(* IEC 61131-3 sources: volt/packages/volt-lsp-iec/test-corpus/pro2193/Device/Plc Logic/Application/09 Misc/Library Manager/L_MC1P_MotionControlBasic (part 2) *)

(* ---- _AXIS_REF_ENC.pou ---- *)
FUNCTION_BLOCK _AXIS_REF_ENC EXTENDS _AXIS_REF_COM
VAR_INPUT
	DIENCODERPOSITION : DINT;
	XENCODERPOSVALID : BOOL := TRUE;
	POSSIGNALPROCESSING : L_MC1P_IPosSignalProcessing;
END_VAR
VAR
	WENCFILTERCYCLES : WORD := 1;
	WENCFILTERCYCLESPOS : WORD := 1;
	VELFILTER : L_MC1P_MeanValueFilter;
	ENCODERCONV : L_MC1P_EncoderConv;
	UDITOTALMEASURINGRANGE : UDINT := 4294967295;
	OPTPOSQUANT : L_MC1P_OptimizePosQuantisation;
	EXTRAPOLATION : L_MC1P_Extra_Interpolation;
	LRSETVALDELAYTIME : LREAL := 0;
	ECOMPENSATIONMODE : L_MC1P_CompensationMode := L_MC1P_CompensationMode.Off;
	XISABSOLUTEENCODER : BOOL := FALSE;
	XDRIVEENABLEDINTERN : BOOL;
	USIHOMEPOSPERMANTENTSETOLD : USINT;
	XHOMEPOSPERMANTENTSETFROMINTERN : BOOL;
	XENCODERPOSVALIDOLD : BOOL;
	XENCODERPOSVALIDINT : BOOL;
	XRESETENCODERPOSHANDLING : BOOL;
	WMICSECTICKSACT : WORD;
	WMICSECTICKSOLD : WORD;
	DIVELEXACT : DINT;
	XABSENCAVAILABLE : BOOL := FALSE;
	DWABSTIMERINFASTINPUTRESOLUTION : DWORD;
	XMANIPULATEABSCOUNTER : BOOL := FALSE;
	XCOUNTEROVERFLOW : BOOL;
	LRSCALEUNITTOPOSOLD : LREAL;
	XORIENTATIONINVACTOLD : BOOL;
	SCHOMEPARAMETER_LROFFSETPOSITIONOLD : LREAL;
	XMAXVELEXCEEDED : BOOL;
	XMAXVELEXCEEDEDOLD : BOOL;
	ITFENCODERPOSFILTER : L_MC1P_IEncoderPosFilter;
	ITFENCODERPOSFILTEROLD : L_MC1P_IEncoderPosFilter;
	ITFENCODERPOSFILTEREXTERNAL : L_MC1P_IEncoderPosFilter;
	FB_MEANPOSFILTER : L_MC1P_MeanEncoderPositionFilter;
	FB_BUTTERWORTHPOSFILTER : L_MC1P_ButterworthEncoderPosFilter;
	LRBTWFILTERTIME : LREAL;
	EENCINPUTFILTER : USINT;
	WENCFILTERCYCLESACTIVE : WORD;
	DIBTWFILTERTIME : DINT;
	EENCPOSFILTERSTATE : WORD;
	EENCVELFILTERSTATE : WORD;
	WENCODERPOSHANDLING : WORD;
	XTIMESTAMPFORPOSSUPPORTED : BOOL;
	_PTASKMAPLIST : POINTER TO IoStandard.IoConfigTaskMap;
	_NTASKMAPLISTCOUNT : DINT;
	_WMODULETYPE : UINT;
	_DWINSTANCE : UDINT;
	_CONNECTOR : POINTER TO IoConfigConnector;
	EENCODERTYPE : L_Mc1P_EncoderType;
	DIINPUTPOSOLD : DINT;
	DIACTPOSUNFILTERED : DINT;
	LRRESIDUALPOSUNFILTERED : LREAL;
	XCONFIGCHANGED : BOOL;
	DWPOSTIMESTAMP : DWORD;
	POSSIGNALPROCESSINGINT : L_MC1P_PosSignalProcessing;
	XSSIENCODER : BOOL := FALSE;
	DWENCODERUPDATETIME : DWORD;
	DIACTPOS1616 : DINT;
	XACTVELFROMPOS : BOOL;
	PDWABSOLUTECOUNTERINT : POINTER TO DWORD;
	DIACTPOSRAWOLD : DINT;
	XVELEXACTSUPPORTED : BOOL;
	CMPID_CMP_LSMCFREEENCODER : DWORD := 16#1028200D;
	ENCHOMEPOSPERMANTENTSETACTIVE : BOOL;
	GETTIMEREFVALUE : DWORD;
	HOMEPOSPERMANTENTSETACTIVE : BOOL;
	WAITFORAXISDETECTION : BOOL;
END_VAR
END_FUNCTION_BLOCK

METHOD CALCACTPOSFROMHWCOUNTER : LREAL
END_METHOD

METHOD CALCACTPOSUNFILTERED : LREAL
END_METHOD

METHOD CALCACTVALUES
END_METHOD

METHOD CALCEXTRAPOLATIONVALUES
VAR_INPUT
	LRACTPOSIN : LREAL;
	LRACTVELIN : LREAL;
	LRACTACCIN : LREAL;
	LRACTTORQUEIN : LREAL;
END_VAR
VAR_OUTPUT
	LRACTPOSOUT : LREAL;
	LRACTVELOUT : LREAL;
	LRACTACCOUT : LREAL;
	LRACTTORQUEOUT : LREAL;
END_VAR
END_METHOD

METHOD CALLRECIEVEPARAMETER
END_METHOD

METHOD CHECKPLAUSIBILITYOFACTVALUES
END_METHOD

METHOD ENCODERSIGNALHANDLING : BOOL
END_METHOD

METHOD GETACTVELOCITYEXACT : LREAL
END_METHOD

METHOD PREPAREINPUTDATA : BOOL
END_METHOD

METHOD READENCODERINPUT : BOOL
VAR_INPUT
	DINEWENCPOS : DINT;
END_VAR
END_METHOD

METHOD RESETACTPOS
END_METHOD

METHOD RESETAXISCONNECTOR
END_METHOD

METHOD RESETENCODERVALUES
END_METHOD

METHOD SETENCODERFILTERINTERFACE
VAR_INPUT
	IENCODERFILTERITF : L_MC1P_IEncoderPosFilter;
END_VAR
END_METHOD

METHOD SETHOMEPOSITION2
VAR_INPUT
	POSITION : LREAL;
	RELATIVE : BOOL;
	XRESTARTPOSITIONING : BOOL := FALSE;
	EHOMEPOSINFO : L_IE1P_Error;
END_VAR
END_METHOD

METHOD ENCNEWHOMEPOSLOADED : BOOL
VAR_INPUT
	DWCALLYCLE : DWORD;
	DWDELAY : DWORD;
END_VAR
END_METHOD

METHOD ENCRESETACTPOS
END_METHOD

METHOD ENCRESETHOMEPOS
VAR_INPUT
	ERESETINFO : L_IE1P_Error;
END_VAR
END_METHOD

METHOD ENCSETHOMEPOSITION
VAR_INPUT
	POSITION : LREAL;
	RELATIVE : BOOL;
	POSDIFF : LREAL;
	EHOMEPOSINFO : L_IE1P_Error;
END_VAR
END_METHOD

METHOD ENCSIGNALVALID : BOOL
VAR_OUTPUT
	XSIGNALVALIDOLD : BOOL;
	EENCERRORID : L_IE1P_Error;
END_VAR
END_METHOD

METHOD GETACTPOSINCR : DINT
END_METHOD

METHOD GETACTPOSINCR1616 : DINT
END_METHOD

METHOD GETACTVALUES
VAR_OUTPUT
	LRACTPOS : LREAL;
	LRACTVEL : LREAL;
	LRACTACC : LREAL;
	LRACTPOSUNFILTERED : LREAL;
	LRACTPOSROUNDS : LREAL;
END_VAR
END_METHOD

METHOD GETAXISINSTANCE : POINTER TO _AXIS_REF_REAL
END_METHOD

METHOD GETCONFIGCHANGED : BOOL
END_METHOD

METHOD GETENCODERINTERFACE : L_MC1P_IEncoderInterface
END_METHOD

METHOD GETHOMEPOSAVAILABLE : BOOL
END_METHOD

METHOD SETHOMEPOSAVAILABLE
VAR_INPUT
	XHOMEPOSAVAILABLE : BOOL;
END_VAR
END_METHOD

METHOD GETVIRTUAL : BOOL
END_METHOD

METHOD CALCSCALEFUNCTIONS
VAR_INPUT
	OFFSET : DWORD;
	INDEX : WORD;
END_VAR
END_METHOD

METHOD CALLTRANSMITPARAMETER
END_METHOD

METHOD PDCONVACTPOS : DINT
VAR_INPUT
	DIINPUT : DINT;
END_VAR
END_METHOD

METHOD PDCONVACTPOSENCCONV : DINT
VAR_INPUT
	DIINPUT : DINT;
END_VAR
END_METHOD

METHOD PDCONVACTVEL : DINT
VAR_INPUT
	DIINPUT : DINT;
END_VAR
END_METHOD

METHOD PDHANDLETIMESTAMPS : DINT
VAR_INPUT
	WMICSECTICK : WORD;
END_VAR
END_METHOD

METHOD CONFIGUREAXIS
END_METHOD

METHOD CONNECTMOTIONUTILS
VAR_INPUT
	DRIVEUTILS : L_MC1P_IDriveUtils;
	AXISEXTENSION : L_MC1P_IAxisExtension;
END_VAR
END_METHOD

METHOD CALCAFTERREADINPUTS : INT
END_METHOD

METHOD CALCBEFOREREADINPUTS : INT
END_METHOD

METHOD CALCBEFOREWRITEOUTPUTS : INT
END_METHOD

METHOD FB_INIT : BOOL
VAR_INPUT
	BINITRETAINS : BOOL;
	BINCOPYCODE : BOOL;
END_VAR
END_METHOD

METHOD IODRVUPDATEMAPPING : UDINT
VAR_INPUT
	PTASKMAPLIST : POINTER TO IoConfigTaskMap;
	NCOUNT : DINT;
END_VAR
END_METHOD

METHOD INITIALIZE : UDINT
VAR_INPUT
	WMODULETYPE : UINT;
	DWINSTANCE : UDINT;
	PCONNECTOR : POINTER TO IoConfigConnector;
END_VAR
END_METHOD

(* ---- _AXIS_REF_ENC_BPB.pou ---- *)
FUNCTION_BLOCK _AXIS_REF_ENC_BPB EXTENDS _AXIS_REF_ENC
VAR
	AXISEXTENSION : L_MC1P_AxisExtension_EncBPB;
	MOTIONUTILS : L_MC1P_MotionUtils_EncBPB;
END_VAR
END_FUNCTION_BLOCK

METHOD FB_INIT : BOOL
VAR_INPUT
	BINITRETAINS : BOOL;
	BINCOPYCODE : BOOL;
END_VAR
END_METHOD

(* ---- _AXIS_REF_ENC_FREE.pou ---- *)
FUNCTION_BLOCK _AXIS_REF_ENC_FREE EXTENDS _AXIS_REF_ENC
VAR
	AXISEXTENSION : L_MC1P_AxisExtension_EncFree;
	MOTIONUTILS : L_MC1P_MotionUtils_EncFree;
END_VAR
END_FUNCTION_BLOCK

METHOD FB_INIT : BOOL
VAR_INPUT
	BINITRETAINS : BOOL;
	BINCOPYCODE : BOOL;
END_VAR
END_METHOD

(* ---- _AXIS_REF_ENC_I500_ECAT.pou ---- *)
FUNCTION_BLOCK _AXIS_REF_ENC_I500_ECAT EXTENDS _AXIS_REF_ENC
VAR
	AXISEXTENSION : L_MC1P_AxisExtension_Enci500;
	MOTIONUTILS : L_MC1P_MotionUtils_Enci500;
END_VAR
END_FUNCTION_BLOCK

METHOD FB_INIT : BOOL
VAR_INPUT
	BINITRETAINS : BOOL;
	BINCOPYCODE : BOOL;
END_VAR
END_METHOD

(* ---- _AXIS_REF_ENC_I900.pou ---- *)
FUNCTION_BLOCK _AXIS_REF_ENC_I900 EXTENDS _AXIS_REF_ENC
END_FUNCTION_BLOCK

METHOD HLP_INITPARREF
END_METHOD

METHOD HLP_READPARAMETER : BOOL
VAR_INPUT
	PARAMETER : DINT;
	PLRVALUE : POINTER TO LREAL;
END_VAR
END_METHOD

(* ---- _AXIS_REF_ENC_I900_CIA.pou ---- *)
FUNCTION_BLOCK _AXIS_REF_ENC_I900_CIA EXTENDS _AXIS_REF_ENC_i900_Target
END_FUNCTION_BLOCK

METHOD SETDRIVECONFIG
VAR_OUTPUT
	XDONE : BOOL;
	XERROR : BOOL;
	WERRORID : WORD;
END_VAR
END_METHOD

METHOD CALCULATESCALING : BOOL
END_METHOD

METHOD FB_INIT : BOOL
VAR_INPUT
	BINITRETAINS : BOOL;
	BINCOPYCODE : BOOL;
END_VAR
END_METHOD

(* ---- _AXIS_REF_ENC_I900_ECAT.pou ---- *)
FUNCTION_BLOCK _AXIS_REF_ENC_I900_ECAT EXTENDS _AXIS_REF_ENC
VAR
	AXISEXTENSION : L_MC1P_AxisExtension_Enci900_ECAT;
	MOTIONUTILS : L_Mc1P_MotionUtils_Enci900_ECAT;
	RETAINMANAGEMENT : L_MC1P_MotionUtilsRetainHandling;
END_VAR
END_FUNCTION_BLOCK

METHOD FB_INIT : BOOL
VAR_INPUT
	BINITRETAINS : BOOL;
	BINCOPYCODE : BOOL;
END_VAR
END_METHOD

(* ---- _AXIS_REF_ENC_I900_TARGET.pou ---- *)
FUNCTION_BLOCK _AXIS_REF_ENC_I900_TARGET EXTENDS _AXIS_REF_ENC_i900
VAR
	AXISEXTENSION : L_MC1P_AxisExtension_Enci900_Target;
	MOTIONUTILS : L_MC1P_MotionUtils_Enci900_Target;
	RETAINMANAGEMENT : L_MC1P_MotionUtilsRetainHandling;
END_VAR
END_FUNCTION_BLOCK

METHOD CALLRECIEVEPARAMETER
END_METHOD

METHOD CONFIGUREAXISCONNECTOR
END_METHOD

METHOD GETIECADRESS
END_METHOD

METHOD FB_INIT : BOOL
VAR_INPUT
	BINITRETAINS : BOOL;
	BINCOPYCODE : BOOL;
END_VAR
END_METHOD

(* ---- _AXIS_REF_ENC_IO_ETC.pou ---- *)
FUNCTION_BLOCK _AXIS_REF_ENC_IO_ETC EXTENDS _AXIS_REF_ENC
VAR
	AXISEXTENSION : L_MC1P_AxisExtension_EncIOEtc;
	MOTIONUTILS : L_MC1P_MotionUtils_EncIOEtc;
END_VAR
END_FUNCTION_BLOCK

METHOD INITIALIZE : UDINT
VAR_INPUT
	WMODULETYPE : UINT;
	DWINSTANCE : UDINT;
	PCONNECTOR : POINTER TO IoConfigConnector;
END_VAR
END_METHOD

METHOD FB_INIT : BOOL
VAR_INPUT
	BINITRETAINS : BOOL;
	BINCOPYCODE : BOOL;
END_VAR
END_METHOD

(* ---- _AXIS_REF_ENC_UNIVERSAL.pou ---- *)
FUNCTION_BLOCK _AXIS_REF_ENC_UNIVERSAL EXTENDS _AXIS_REF_ENC
VAR
	FBDRIVESPECIFIC : L_MC1P_DriveSpecific_Enc_Free;
	AXISEXTENSIONFACTORY : L_MC1P_UniversalEncoderFactory;
	ITFDRIVEUTILSTOCONNECT : POINTER TO L_MC1P_IDriveUtils;
	ITFAXISEXTENSION : L_MC1P_IAxisExtension;
	UITYPE : UINT := 2;
	DRIVESPECIFICBASIC : L_MC1P_IDriveSpecificImplBase;
	WAITFORAXISDETECTION : BOOL;
END_VAR
END_FUNCTION_BLOCK

METHOD CALCAFTERREADINPUTS : INT
END_METHOD

METHOD CONNECTASYNC : BOOL
END_METHOD

METHOD CREATEAXISEXTENSION : L_MC1P_IAxisExtension
VAR_INPUT
	EAXISEXTENSIONTYPE : L_MC1P_AxisExtensionTypes;
END_VAR
END_METHOD

METHOD DISCONNECTMOTIONUTILS : BOOL
VAR_INPUT
	EDISCONNECTMODE : L_IF1P_DisconnectMode;
END_VAR
END_METHOD

METHOD FINDANDCONNECTMOTIONUTILS
END_METHOD

METHOD FINDDRIVEUTILSINMOTIONCONNECTOR : BOOL
VAR_INPUT
	PECATSLAVECONNECTOR : POINTER TO IoConfigConnector;
	SUBDEVICE : UINT;
END_VAR
END_METHOD

METHOD INITIALIZE : UDINT
VAR_INPUT
	WMODULETYPE : UINT;
	DWINSTANCE : UDINT;
	PCONNECTOR : POINTER TO IoConfigConnector;
END_VAR
END_METHOD

METHOD FB_INIT : BOOL
VAR_INPUT
	BINITRETAINS : BOOL;
	BINCOPYCODE : BOOL;
END_VAR
END_METHOD

METHOD CONNECTDEVICE : UINT
VAR_INPUT
	DEVICEMODULEHANDLER : L_IMHP_IModuleHandler;
	UISUBDEVICE : UINT := 0;
	EDISCONNECTMODE : L_IF1P_DisconnectMode;
	XDISCONNECTEXISTINGCONNECTION : BOOL;
END_VAR
VAR_OUTPUT
	ITFCONNECTIONFBSTATUS : L_IF1P_IStatus;
END_VAR
END_METHOD

METHOD DISCONNECTDEVICE : UINT
VAR_INPUT
	EDISCONNECTMODE : L_IF1P_DisconnectMode;
	XBUSYBEFORE : BOOL;
END_VAR
VAR_OUTPUT
	ITFCONNECTIONFBSTATUS : L_IF1P_IStatus;
END_VAR
END_METHOD

METHOD GEFUNCTIONTINSTANCEPOINTER : POINTER TO BYTE
END_METHOD

METHOD GETCONNECTEDDEVICE : L_IMHP_IModuleHandler
VAR_OUTPUT
	UISUBDEVICE : UINT := 0;
	XVALID : BOOL;
	ITFCONNECTIONFBSTATUS : L_IF1P_IStatus;
END_VAR
END_METHOD

METHOD GETCONNECTIONDIAGNOSTIC
VAR_OUTPUT
	WUSEDBY_COMP : WORD;
	WUSEDBY_SUBCOMP : WORD;
	WACTIVEMODE : WORD;
	WSUBDEVICE : WORD;
	SCONNECTIONSOURE : STRING;
END_VAR
END_METHOD

METHOD GETITFCONNECTSTATUS
VAR_OUTPUT
	ITFCONNECTIONFBSTATUS : L_IF1P_IStatus;
END_VAR
END_METHOD

(* ---- _AXIS_REF_GENERIC.pou ---- *)
FUNCTION_BLOCK _AXIS_REF_GENERIC EXTENDS _AXIS_REF_COM
VAR
	AXISEXTENSION : L_MC1P_AxisExtension_GenericDrive;
	MOTIONUTILS : L_MC1P_MotionUtils_GenericDrive;
	RETAINMANAGEMENT : L_MC1P_MotionUtilsRetainHandling;
END_VAR
END_FUNCTION_BLOCK

METHOD SETGENERICCONFIGURATION
VAR_INPUT
	ITFGENERICCONFIG : L_MC1P_IGenericAxisConfiguration;
END_VAR
END_METHOD

METHOD FB_INIT : BOOL
VAR_INPUT
	BINITRETAINS : BOOL;
	BINCOPYCODE : BOOL;
END_VAR
END_METHOD

(* ---- _AXIS_REF_I500.pou ---- *)
FUNCTION_BLOCK _AXIS_REF_I500 EXTENDS _AXIS_REF_COM
VAR
	CONFIGAXIS : L_MC1P_Config_i500;
	FBEXTENDEDMAPPINGACCESS : L_MC1P_ExtendedMappingAccess;
	BRAKE : L_MC1P_BrakeControl;
	WNETWORDIN1 : REFERENCE TO WORD;
	WNETWORDIN2 : REFERENCE TO WORD;
	WNETWORDIN3 : REFERENCE TO WORD;
	WNETWORDIN4 : REFERENCE TO WORD;
	WNETWORDOUT1 : REFERENCE TO WORD;
	WNETWORDOUT2 : REFERENCE TO WORD;
	PXDUMMY : POINTER TO BOOL;
	XENABLEDRIVEOLD : BOOL;
	XDEACTIVATEPOSCTRLEXTENCERROR : BOOL;
	NETWORDIN1 : WORD;
	NETWORDIN2 : WORD;
	NETWORDIN3 : WORD;
	NETWORDIN4 : WORD;
	NETWORDOUT1 : WORD;
	NETWORDOUT2 : WORD;
END_VAR
END_FUNCTION_BLOCK

(* ---- _AXIS_REF_I500_CAN.pou ---- *)
FUNCTION_BLOCK _AXIS_REF_I500_CAN EXTENDS _AXIS_REF_i500
VAR
	AXISEXTENSION : L_MC1P_AxisExtension_i500_CAN;
	MOTIONUTILS : L_MC1P_MotionUtils_i500_CAN;
END_VAR
END_FUNCTION_BLOCK

METHOD FB_INIT : BOOL
VAR_INPUT
	BINITRETAINS : BOOL;
	BINCOPYCODE : BOOL;
END_VAR
END_METHOD

(* ---- _AXIS_REF_I500_ETC.pou ---- *)
FUNCTION_BLOCK _AXIS_REF_I500_ETC EXTENDS _AXIS_REF_i500
VAR
	AXISEXTENSION : L_MC1P_AxisExtension_i500_ECAT;
	MOTIONUTILS : L_MC1P_MotionUtils_i500_ECAT;
END_VAR
END_FUNCTION_BLOCK

METHOD FB_INIT : BOOL
VAR_INPUT
	BINITRETAINS : BOOL;
	BINCOPYCODE : BOOL;
END_VAR
END_METHOD

(* ---- _AXIS_REF_I700.pou ---- *)
FUNCTION_BLOCK _AXIS_REF_I700 EXTENDS _AXIS_REF_COM
VAR
	XSLOT2 : BOOL;
	AXISEXTENSION : L_MC1P_AxisExtension_i700;
	MOTIONUTILS : L_MC1P_MotionUtils_i700;
	RETAINMANAGEMENT : L_MC1P_MotionUtilsRetainHandling;
END_VAR
END_FUNCTION_BLOCK

METHOD INITIALIZE : UDINT
VAR_INPUT
	WMODULETYPE : UINT;
	DWINSTANCE : UDINT;
	PCONNECTOR : POINTER TO IoConfigConnector;
END_VAR
END_METHOD

METHOD FB_INIT : BOOL
VAR_INPUT
	BINITRETAINS : BOOL;
	BINCOPYCODE : BOOL;
END_VAR
END_METHOD

(* ---- _AXIS_REF_I700_SLOT1.pou ---- *)
FUNCTION_BLOCK _AXIS_REF_I700_SLOT1 EXTENDS _AXIS_REF_i700
END_FUNCTION_BLOCK

METHOD FB_INIT : BOOL
VAR_INPUT
	BINITRETAINS : BOOL;
	BINCOPYCODE : BOOL;
END_VAR
END_METHOD

(* ---- _AXIS_REF_I750.pou ---- *)
FUNCTION_BLOCK _AXIS_REF_I750 EXTENDS _AXIS_REF_COM
VAR
	XSLOT2 : BOOL;
	AXISEXTENSION : L_MC1P_AxisExtension_i750;
	MOTIONUTILS : L_MC1P_MotionUtils_i750;
	RETAINMANAGEMENT : L_MC1P_MotionUtilsRetainHandling;
END_VAR
END_FUNCTION_BLOCK

METHOD FB_INIT : BOOL
VAR_INPUT
	BINITRETAINS : BOOL;
	BINCOPYCODE : BOOL;
END_VAR
END_METHOD

(* ---- _AXIS_REF_I900.pou ---- *)
FUNCTION_BLOCK _AXIS_REF_I900 EXTENDS _AXIS_REF_COM
VAR
	XSLOT2 : BOOL;
	AXISEXTENSION : L_MC1P_AxisExtension_i950;
	MOTIONUTILS : L_MC1P_MotionUtils_i950;
	RETAINMANAGEMENT : L_MC1P_MotionUtilsRetainHandling;
END_VAR
END_FUNCTION_BLOCK

METHOD FB_INIT : BOOL
VAR_INPUT
	BINITRETAINS : BOOL;
	BINCOPYCODE : BOOL;
END_VAR
END_METHOD

(* ---- _AXIS_REF_I900_CIAADV.pou ---- *)
FUNCTION_BLOCK _AXIS_REF_I900_CIAADV EXTENDS _AXIS_REF_COM
VAR
	XSLOT2 : BOOL;
	AXISEXTENSION : L_MC1P_AxisExtension_i950_CiaAdv;
	MOTIONUTILS : L_MC1P_MotionUtils_i950_CiaAdv;
	RETAINMANAGEMENT : L_MC1P_MotionUtilsRetainHandling;
END_VAR
END_FUNCTION_BLOCK

METHOD FB_INIT : BOOL
VAR_INPUT
	BINITRETAINS : BOOL;
	BINCOPYCODE : BOOL;
END_VAR
END_METHOD

(* ---- _AXIS_REF_I900_DRIVE.pou ---- *)
FUNCTION_BLOCK _AXIS_REF_I900_DRIVE EXTENDS _AXIS_REF_COM
VAR
	LRHOMETORQUELIMIT : LREAL;
	LRHOMETORQUELIMITTIME : LREAL;
	EFOLLOWINGERRORREACTIONI900 : USINT;
	XIGNOREPDOINTERFACEDISABLED : BOOL := FALSE;
	INTERPOLATION : L_MC1P_DelaySetValues2;
	LRSETVALDELAYTIME : LREAL := 0;
	ECOMPENSATIONMODE : L_MC1P_CompensationMode := L_MC1P_CompensationMode.Off;
	UIPOSCTRLADAPTACTIVEVALUE : UINT;
	USIPOSCTRLADAPTIONFROM0X2985 : USINT := 0;
	POSCTRLADAPTIONCURVE : L_MC1P_PosCtrlAdaptionCurve;
	DWCOMPATIBILITYFLAGS_0X2DE0_28 : DWORD;
	WAITFORAXISDETECTION : BOOL;
END_VAR
END_FUNCTION_BLOCK

METHOD GETACTIVEPOSCTRLADAPTVALUE : LREAL
END_METHOD

METHOD CONFIGUREAXISCONNECTOR
END_METHOD

METHOD CALCSCALEFUNCTIONS
VAR_INPUT
	OFFSET : DWORD;
	INDEX : WORD;
END_VAR
END_METHOD

METHOD UPDATEDRIVEOFFSETHANDLING
VAR_INPUT
	DWACTCYCLECOUNTERVALUE : DWORD;
	XRESET : BOOL;
END_VAR
END_METHOD

METHOD HLP_INITPARREF
END_METHOD

METHOD HLP_READBOOLPARAMETER : BOOL
VAR_INPUT
	PARAMETER : DINT;
	PXVALUE : POINTER TO BOOL;
END_VAR
END_METHOD

METHOD HLP_READPARAMETER : BOOL
VAR_INPUT
	PARAMETER : DINT;
	PLRVALUE : POINTER TO LREAL;
END_VAR
END_METHOD

METHOD HLP_WRITEBOOLPARAMETER : BOOL
VAR_INPUT
	PARAMETER : DINT;
	PXVALUE : POINTER TO BOOL;
END_VAR
VAR_OUTPUT
	WERRORID : WORD;
END_VAR
END_METHOD

METHOD CALCBEFOREREADINPUTS : INT
END_METHOD

METHOD CALCBEFOREWRITEOUTPUTS : INT
END_METHOD

METHOD FB_INIT : BOOL
VAR_INPUT
	BINITRETAINS : BOOL;
	BINCOPYCODE : BOOL;
END_VAR
END_METHOD

(* ---- _AXIS_REF_I900_DRIVE_CIA.pou ---- *)
FUNCTION_BLOCK _AXIS_REF_I900_DRIVE_CIA EXTENDS _AXIS_REF_i900_Drive_Target
VAR_INPUT
	XOPMODEVIACIA402INTERFACE : BOOL;
	XCONTROLVIACIAINTERFACE : BOOL;
	XSETVALUESVIAAPPLICATION : BOOL;
	CIA_CTRL_EXT : WORD;
	CIA_OPMOD_EXT : SINT;
	WLENZECTRL_EXT : WORD;
	WTPCONTROL12 : WORD;
	WTPCONTROL34 : WORD;
	XCONTROLVIACIAINTERFACEOLD : BOOL;
	XEXTSETVALUESVALID : BOOL;
	LRSETPOSITION_EXT : LREAL;
	LRSETVELOCITY_EXT : LREAL;
	LRSETTORQUE_EXT : LREAL;
	LRSETVELOCITYLIMITHIGH_EXT : LREAL;
	LRSETVELOCITYLIMITLOW_EXT : LREAL;
	LRSETVLVELOCITY_EXT : LREAL;
END_VAR
VAR_OUTPUT
	WTPSTATUS12 : WORD;
	WTPSTATUS34 : WORD;
	LRTP1_POSEDGE : LREAL;
	LRTP1_NEGEDGE : LREAL;
	DWTP1_TIMENEGEDGE : DWORD;
	DWTP1_TIMEPOSEDGE : DWORD;
	LRTP2_POSEDGE : LREAL;
	LRTP2_NEGEDGE : LREAL;
	DWTP2_TIMENEGEDGE : DWORD;
	DWTP2_TIMEPOSEDGE : DWORD;
	LRTP3_POSEDGE : LREAL;
	LRTP3_NEGEDGE : LREAL;
	DWTP3_TIMENEGEDGE : DWORD;
	DWTP3_TIMEPOSEDGE : DWORD;
	LRTP4_POSEDGE : LREAL;
	LRTP4_NEGEDGE : LREAL;
	DWTP4_TIMENEGEDGE : DWORD;
	DWTP4_TIMEPOSEDGE : DWORD;
	LRACTCONTROLEFFORT : LREAL;
END_VAR
VAR
	WPOWID : WORD;
	CIA_CTRLOLD_EXT : WORD;
	XSETVALUESVIAAPPLICATION_INT : BOOL;
	XINTTP1ACTIVE : BOOL;
	XINTTP2ACTIVE : BOOL;
	XINTTP3ACTIVE : BOOL;
	XINTTP4ACTIVE : BOOL;
	DIDRIVEREFOFFSET : DINT;
	DIDRIVEREFOFFSETABS : DINT;
	DIDRIVEREFOFFSETABSOLD : DINT;
	XDRIVELOADPOS : BOOL;
	XIGNOREDRIVEOFFSET : BOOL;
	DIDEBUGPOS : DINT;
	REFOFFSETHANDLING : L_MC1P_i900RefOffsetHandling;
	XREFOFFSETHANDLINGCALCULATED : BOOL;
	XCONFIGCHANGED : BOOL;
	XCONFIGCHANGEDENCODER : BOOL;
	X2NDFDBACTIVE : BOOL;
	X2NDFDBOBSERVATIONACTIVE : BOOL;
	LRDIRECTIONHYSTERESISDIFFOLD : LREAL;
	LRACTCONTROLEFFORTDRIVE : LREAL;
	WLENZECTRL : REFERENCE TO WORD;
	LRSPEEDCTRLINT : REFERENCE TO LREAL;
	XNEWHOMEPOSHANDLINGCIA402ADV : BOOL;
	CIA402ADVANCEDAXIS : BOOL;
	STARTPOSFORINTERNALSTOP : LREAL;
END_VAR
END_FUNCTION_BLOCK

METHOD CALCACTVALUES
END_METHOD

METHOD CALCCONTOLLER
END_METHOD

METHOD CALCDRIVEHOMEOFFSET : DINT
VAR_INPUT
	LROLDPOS : LREAL;
	LRNEWPOSPOS : LREAL;
END_VAR
END_METHOD

METHOD CHECKFOLLOWINGERROR : BOOL
END_METHOD

METHOD CHECKPLNOTVALID : BOOL
END_METHOD

METHOD CONVERTTPPOSAPP : LREAL
VAR_INPUT
	DIPOS : DINT;
END_VAR
END_METHOD

METHOD ENABLEDRIVE : BOOL
VAR_INPUT
	XENABLE : BOOL;
END_VAR
END_METHOD

METHOD GETACTDIRECTION : MC_DIRECTION
VAR_INPUT
	XCALCULATE : BOOL;
END_VAR
END_METHOD

METHOD GETDRIVESTATE : BOOL
END_METHOD

METHOD HANDLETPCONTROL
VAR_INPUT
	WTPCONTROL : WORD;
	PWCONTROL : POINTER TO WORD;
END_VAR
VAR_IN_OUT
	XTP1ACTIVE : BOOL;
	XTP2ACTIVE : BOOL;
END_VAR
END_METHOD

METHOD RESETACTPOS
END_METHOD

METHOD RESETCONFIGCHANGED
END_METHOD

METHOD SETHOMEPOSITION2
VAR_INPUT
	POSITION : LREAL;
	RELATIVE : BOOL;
	XRESTARTPOSITIONING : BOOL := FALSE;
	EHOMEPOSINFO : L_IE1P_Error;
END_VAR
END_METHOD

METHOD PDCONVACTPOS : DINT
VAR_INPUT
	DIINPUT : DINT;
END_VAR
END_METHOD

METHOD PDCONVSETPOS : DINT
VAR_INPUT
	XSETEQACTONDISABLED : BOOL;
END_VAR
END_METHOD

METHOD PDCONVTPPOS : DINT
VAR_INPUT
	DIPOS : DINT;
END_VAR
END_METHOD

METHOD SETDRIVECONFIG
VAR_OUTPUT
	XDONE : BOOL;
	XERROR : BOOL;
	WERRORID : WORD;
END_VAR
END_METHOD

METHOD CALCPOSTOUNIT : LREAL
VAR_INPUT
	DIPOSITION : DINT;
END_VAR
END_METHOD

METHOD CALCRPMTOUNIT : LREAL
VAR_INPUT
	ISPEED : INT;
END_VAR
END_METHOD

METHOD CALCSPEEDTOUNIT : LREAL
VAR_INPUT
	DISPEED : DINT;
END_VAR
END_METHOD

METHOD CALCTORQUETOUNIT : LREAL
VAR_INPUT
	ITORQUE : INT;
END_VAR
END_METHOD

METHOD CALCUNITTOPOS : DINT
VAR_INPUT
	LRPOSITION : LREAL;
END_VAR
END_METHOD

METHOD CALCUNITTORPM : INT
VAR_INPUT
	LRVELOCITY : LREAL;
END_VAR
END_METHOD

METHOD CALCUNITTOSPEED : DINT
VAR_INPUT
	LRVELOCITY : LREAL;
END_VAR
END_METHOD

METHOD CALCUNITTOTORQUE : INT
VAR_INPUT
	LRTORQUE : LREAL;
END_VAR
END_METHOD

METHOD CALCULATESCALING : BOOL
END_METHOD

METHOD RESTOREACTPOS
VAR_INPUT
	PPOSDATA : POINTER TO L_MC1P_uRetainData;
END_VAR
END_METHOD

METHOD RETAINHANDLING : BOOL
END_METHOD

METHOD STOREACTPOS
VAR_INPUT
	PPOSDATA : POINTER TO L_MC1P_uRetainData;
END_VAR
END_METHOD

METHOD STOREADDITIONALRETAINDATA
VAR_INPUT
	PDATA : POINTER TO L_MC1P_uRetainData;
END_VAR
END_METHOD

METHOD CALCBEFOREREADINPUTS : INT
END_METHOD

METHOD GETIECADRESS
END_METHOD

METHOD RECEIVEPARAMETER2
VAR_INPUT
	WPARAMETER : WORD;
	PADRESS : POINTER TO BYTE;
	WSIZE : WORD;
	PADDDATA : POINTER TO L_SI9P_IODrvMappingData;
END_VAR
END_METHOD

METHOD RECEIVEPARAMETERCALC2
VAR_IN_OUT
	DATA : ARRAY [1..L_MC1P_Constants.gc_Rec_MaxDataIndex] OF POINTER TO L_MC1P_MappedElement;
END_VAR
END_METHOD

METHOD TRANSMITPARAMETER
VAR_INPUT
	WPARAMETER : WORD;
	PADRESS : POINTER TO BYTE;
	WSIZE : WORD;
END_VAR
END_METHOD

METHOD TRANSMITPARAMETER2
VAR_INPUT
	WPARAMETER : WORD;
	PADRESS : POINTER TO BYTE;
	WSIZE : WORD;
	PADDDATA : POINTER TO L_SI9P_IODrvMappingData;
END_VAR
END_METHOD

METHOD TRANSMITPARAMETERCALC2
VAR_IN_OUT
	DATA : ARRAY [1..L_MC1P_Constants.gc_Trans_MaxDataIndex] OF POINTER TO L_MC1P_MappedElement;
END_VAR
END_METHOD

METHOD FB_INIT : BOOL
VAR_INPUT
	BINITRETAINS : BOOL;
	BINCOPYCODE : BOOL;
END_VAR
END_METHOD

(* ---- _AXIS_REF_I900_DRIVE_TARGET.pou ---- *)
FUNCTION_BLOCK _AXIS_REF_I900_DRIVE_TARGET EXTENDS _AXIS_REF_i900_Drive
VAR
	AXISEXTENSION : L_MC1P_AxisExtension_i950_Drive;
	MOTIONUTILS : L_MC1P_MotionUtils_i950_Drive;
	RETAINMANAGEMENT : L_MC1P_MotionUtilsRetainHandling;
	ADWINTERNALMAPPEDWRITEOBJECTS : ARRAY [1..c_wMaxTransElem] OF DWORD;
	HEVENTSETERRORREACTION : SysTypes.RTS_IEC_HANDLE := SysTypes.RTS_INVALID_HANDLE;
	HINTERFACESETERRORREACTION : SysTypes.RTS_IEC_HANDLE := SysTypes.RTS_INVALID_HANDLE;
	HEVENTUPDATEACTIVEERROR : SysTypes.RTS_IEC_HANDLE := SysTypes.RTS_INVALID_HANDLE;
	HINTERFACEUPDATEACTIVEERROR : SysTypes.RTS_IEC_HANDLE := SysTypes.RTS_INVALID_HANDLE;
	XINITIALREADERRORSTATUS : BOOL := FALSE;
	USIACTIVEERRORINFO : USINT := 0;
	DWLEMERRORCODE : ARRAY [0..2] OF DWORD;
	USILEMSEVERITY : ARRAY [0..2] OF USINT;
	DWPARMONITID : DWORD;
	PIPARQSPOPTION : POINTER TO INT;
	PWPARQSPOPTIONVALID : POINTER TO WORD;
	IPARQSPOPTIONOLD : INT;
	PWPARMOTORRATEDSPEED : POINTER TO WORD;
	PWPARMOTORRATEDSPEEDVALID : POINTER TO WORD;
	WPARMOTORRATEDSPEEDOLD : WORD;
	PDWPARREFTORQUE : POINTER TO DWORD;
	PWPARREFTORQUEVALID : POINTER TO WORD;
	DWPARREFTORQUEOLD : DWORD;
	PDWPARINERTIAMOTOR : POINTER TO DWORD;
	PWPARINERTIAMOTORVALID : POINTER TO WORD;
	DWPARINERTIAMOTOROLD : DWORD;
	PUSIPARMCTRLMODE : POINTER TO USINT;
	PWPARMCTRLMODEVALID : POINTER TO WORD;
	USIPARMCTRLMODEOLD : USINT;
	PDWPARMOTORRATEDCURRENT : POINTER TO DWORD;
	PWPARMOTORRATEDCURRENTVALID : POINTER TO WORD;
	DWPARMOTORRATEDCURRENTOLD : DWORD;
	PDWPARCOMPATIBILITYMODE : POINTER TO DWORD;
	PWPARCOMPATIBILITYMODEVALID : POINTER TO WORD;
	DWPARCOMPATIBILITYMODEOLD : DWORD;
	APWPARGAINADAPTSPEED : ARRAY [1..5] OF POINTER TO WORD;
	APWPARGAINADAPTSPEEDVALID : ARRAY [1..5] OF POINTER TO WORD;
	APWPARGAINADAPTOUT : ARRAY [1..5] OF POINTER TO WORD;
	APWPARGAINADAPTOUTVALID : ARRAY [1..5] OF POINTER TO WORD;
	EQUICKSTOPOPTIONACTIVE : L_MC1P_QuickStopOption := L_MC1P_QuickStopOption.StayInQSP;
END_VAR
END_FUNCTION_BLOCK

METHOD CALCDEPENDENTTORQUEVALUES
VAR_INPUT
	DWDATA : DWORD;
END_VAR
END_METHOD

METHOD GETACTIVEQUICKSTOPOPTION : L_MC1P_QuickStopOption
END_METHOD

METHOD READINITIALREADERRORSTATUS : BOOL
END_METHOD

METHOD CALLRECIEVEPARAMETER
END_METHOD

METHOD CALLTRANSMITPARAMETER
END_METHOD

METHOD CHECKMAPPEDDATAVALID : BOOL
VAR_INPUT
	PADDDATA : POINTER TO BYTE;
	PDATA : POINTER TO POINTER TO BYTE;
END_VAR
VAR_OUTPUT
	XERROR : BOOL;
	EERRORID : L_IE1P_Error;
END_VAR
END_METHOD

METHOD GETMAPPEDDATA : POINTER TO BYTE
VAR_INPUT
	UIINDEX : WORD;
	USISUBINDEX : USINT;
	USISIZE : USINT;
	XWRITEACCESS : BOOL;
	PADDDATA : POINTER TO BYTE;
	PXWAITFORINITACCESS : POINTER TO BOOL;
END_VAR
VAR_OUTPUT
	EERRORID : L_IE1P_Error;
	XERROR : BOOL;
	USISIZEACT : USINT := 0;
END_VAR
END_METHOD

METHOD GETMAPPEDDATASUPPORT : BOOL
END_METHOD

METHOD RECEIVEPARAMETER2
VAR_INPUT
	WPARAMETER : WORD;
	PADRESS : POINTER TO BYTE;
	WSIZE : WORD;
	PADDDATA : POINTER TO L_SI9P_IODrvMappingData;
END_VAR
END_METHOD

METHOD RECEIVEPARAMETERCALC2
VAR_IN_OUT
	DATA : ARRAY [1..L_MC1P_Constants.gc_Rec_MaxDataIndex] OF POINTER TO L_MC1P_MappedElement;
END_VAR
END_METHOD

METHOD RESETMAPPEDDATA
VAR_INPUT
	PADDDATA : POINTER TO BYTE;
END_VAR
END_METHOD

METHOD TRANSMITPARAMETER2
VAR_INPUT
	WPARAMETER : WORD;
	PADRESS : POINTER TO BYTE;
	WSIZE : WORD;
	PADDDATA : POINTER TO L_SI9P_IODrvMappingData;
END_VAR
END_METHOD

METHOD TRANSMITPARAMETERCALC2
VAR_IN_OUT
	DATA : ARRAY [1..L_MC1P_Constants.gc_Trans_MaxDataIndex] OF POINTER TO L_MC1P_MappedElement;
END_VAR
END_METHOD

METHOD EVENTCALLBACK : UDINT
VAR_INPUT
	PEVENTPARAM : POINTER TO EventParam;
END_VAR
END_METHOD

METHOD REGISTEREVENT
END_METHOD

METHOD UNREGISTEREVENT
END_METHOD

METHOD ITFGETACTUALERRORCODE : DWORD
VAR_OUTPUT
	ESEVERITY : WORD;
END_VAR
END_METHOD

METHOD GETIECADRESS
END_METHOD

METHOD FB_INIT : BOOL
VAR_INPUT
	BINITRETAINS : BOOL;
	BINCOPYCODE : BOOL;
END_VAR
END_METHOD

(* ---- _AXIS_REF_REAL.pou ---- *)
FUNCTION_BLOCK _AXIS_REF_REAL EXTENDS AXIS_REF
VAR_OUTPUT
	EACTCONTROLMODE : L_MC1P_ControlMode := 0;
END_VAR
VAR
	DISETPOSTODRIVE : DINT;
	XRESTOREHOMEPOSITION : BOOL := 0;
	XSTORERETAINPOSITION : BOOL := 0;
	LRRESTORETRESHOLD : LREAL := 0;
	SENCODER : STRING;
	PENCODER : POINTER TO BYTE;
	XENCODERSIGNALVALID : BOOL;
	LRPOSCTRLGAIN : LREAL := 20;
	LRPOSCTRLOUTPUTLIMITATION : LREAL := 100000.0;
	XUSEASVIRTUAL : BOOL := 0;
	XUSEASVIRTUALACT : BOOL := 0;
	LRFEEDCONSTANT : LREAL := 360.0;
	DWRATIODEN : DWORD := 1;
	DWRATIONUM : DWORD := 1;
	DWRATIODENADD : DWORD := 1;
	DWRATIONUMADD : DWORD := 1;
	XORIENTATIONINV : BOOL := 0;
	DWINKPERREV : DWORD := 65536;
	LRINERTIALOAD : LREAL := 0.0;
	LRINERTIAMOTOR : LREAL := 0.0;
	LRREFTORQUE : LREAL := 0.0;
	LRMOTORRATEDTORQUEAPP : LREAL := 0.0;
	LRTORQUELIMITDEFAULT : LREAL := 0.0;
	XENABLEFOLLOWINGERROR : BOOL := 0;
	LRMAXFOLLOWINGERROR1 : LREAL := 0.0;
	LRMAXFOLLOWINGERROR2 : LREAL := 0.0;
	EFOLLOWINGERRORREACTION : WORD;
	XFOLLOWINGERRORWARNINGACTIVE : BOOL;
	XFOLLOWINGERRORERRORACTIVE : BOOL;
	RLIMITSWITCHON : REAL := 10.0;
	XINTERNALMAPPINGDONE : BOOL;
	LWTRANSDATA : LWORD;
	WTRANSELEMENTS : WORD;
	ATRANSELEMENT : ARRAY [1..c_wMaxTransElem] OF L_MC1P_MappedElement;
	ATRANSELEMENTADRESS : ARRAY [1..L_MC1P_Constants.gc_Trans_MaxDataIndex] OF POINTER TO L_MC1P_MappedElement;
	WTRANSELEMENTSADD : WORD;
	ATRANSELEMENTADDITIONAL : ARRAY [1..c_wMaxTransElemAdd] OF POINTER TO L_MC1P_MappedElement;
	LWRECDATA : LWORD;
	WRECEIVEELEMENTS : WORD;
	ARECEIVEELEMENT : ARRAY [1..c_wMaxRecElem] OF L_MC1P_MappedElement;
	ARECEIVEELEMENTADRESS : ARRAY [1..L_MC1P_Constants.gc_Rec_MaxDataIndex] OF POINTER TO L_MC1P_MappedElement;
	WRECELEMENTSADD : WORD;
	ARECELEMENTADDITIONAL : ARRAY [1..c_wMaxRecElemAdd] OF POINTER TO L_MC1P_MappedElement;
	DRIVESTATUSBITS : L_MC1P_DriveStateCollection;
	CIA_SETPOS : DINT;
	CIA_SETVEL : DINT;
	CIA_SETTORQUE : DINT;
	CIA_ACTPOS : DINT;
	CIA_ACTVEL : DINT;
	CIA_ACTTORQUE : DINT;
	CIA_ACTPOSRAW : DINT;
	CIA_VLACTVELOCITY : INT;
	CIA_VLTARGETVELOCITY : INT;
	CIA_CTRL : WORD;
	CIA_OPMOD : SINT;
	CIA_STATE : WORD;
	CIA_OPMODACT : SINT;
	CIA_ACTPOSOLD : DINT;
	CIA_ACTVELOLD : DINT;
	UACTPOS : L_MC1P_PosLINT;
	DWDIGITALINPUTS : DWORD;
	BYDRIVESTATE : BYTE;
	DIRESPEEDDIFF : DINT;
	LISETPOSINC : LINT;
	LISETPOSINCOLD : LINT;
	DIREFOFFSETINCDRIVE : DINT;
	DIMTOFFSETINC : DINT;
	LRVLACTVELOCITY : LREAL;
	BYDELAYDRIVEOPERATIONENABLED : BYTE;
	BYDELAYLIMITDRIVEOPERATIONENABLED : BYTE := 2;
	XRESETHOMEPOS : BOOL;
	UIPOSCTRLADAPTVALUE : UINT := 10000;
	POSCONTROLLER : L_MC1P_PosControllerV2;
	ITFPOSCONTROLLER : L_MC1P_IControllerInterface;
	LRSETPOSITIONINT : LREAL;
	LRSETVELOCITYINT : LREAL;
	LRSETACCELERATIONINT : LREAL;
	LRSETTORQUEINT : LREAL;
	LRSETVELOCITYLIMITHIGHINT : LREAL := 0;
	LRSETVELOCITYLIMITLOWINT : LREAL := 0;
	ITFBRAKE : L_MC1P_IAXIS_REF_BRAKE;
	DWREVISION : DWORD;
	DWMOTORRATEDSPEED : DWORD;
	LRMOTORRATEDVELOCITY : LREAL;
	LRMOTORRATEDTORQUE : LREAL;
	DWENCODERCRC : DWORD;
	DWMOTORREVOLUTION : DWORD;
	XNEWHOMEPOSFORENCODERLOADED : BOOL;
	XFEEDBACKABSPOSAVAILABLE : BOOL;
	LRINERTIALOADACT : LREAL;
	LRINERTIAADAPT : LREAL := 1;
	LRFEEDCONSTANTACT : LREAL := 360.0;
	DWRATIONUMACT : DWORD := 1;
	DWRATIODENACT : DWORD := 1;
	DWRATIONUMADDACT : DWORD := 1;
	DWRATIODENADDACT : DWORD := 1;
	DWINKPERREVACT : DWORD := 65536;
	LRINCPERREV : LREAL := 65536.0;
	XWRITEPOSRESOLUTION : BOOL := FALSE;
	XORIENTATIONINVACT : BOOL := FALSE;
	LRREFTORQUEMOTOR : LREAL := 0;
	LRREFTORQUEMOTORACT : LREAL := 0;
	LRREFCURRENTMOTOR : LREAL;
	LREFFGEARFACTOR : LREAL := 1.0;
	LRSCALEPOSTOUNIT : LREAL := 1.0;
	LRSCALEREVTOUNIT : LREAL := 1.0;
	LRSCALERPMTOUNIT : LREAL := 1.0;
	LRSCALESPEEDTOUNIT : LREAL := 1.0;
	LRSCALEACCTOUNIT : LREAL := 1.0;
	LRSCALETORQUETOUNIT : LREAL := 1.0;
	LRSCALEUNITTOPOS : LREAL := 1.0;
	LRSCALEUNITTOREV : LREAL := 1.0;
	LRSCALEUNITTOSPEED : LREAL := 1.0;
	LRSCALEUNITTOACC : LREAL := 1.0;
	LRSCALEUNITTOTORQUE : LREAL := 1.0;
	LRSCALEUNITTORPM : LREAL := 1.0;
	LICYCLELENGTHINCRINT : LINT;
	UDICYCLELENGTHINCRRES : UDINT;
	UDISETPOSRES : UDINT;
	LRSCALETORQUETONORM : LREAL := 1.0;
	LRSCALETORQUETONORM2 : LREAL := 1.0;
	LRSCALENORMTOTORQUE : LREAL := 1.0;
	XACTPOSFROMDRIVE : BOOL := TRUE;
	LRACTPOSITIONDRIVE : LREAL;
	LRACTPOSITIONUNFILTEREDDRIVE : LREAL;
	LRACTVELOCITYDRIVE : LREAL;
	LRACTACCELERATIONDRIVE : LREAL;
	LRACTPOSROUNDSDRIVE : LREAL;
	LRABSREFOFFSETDRIVE : LREAL;
	LRLOADPOSOFFSET : LREAL;
	ERETAINDATATYPE : L_MC1P_RetainDataType := L_MC1P_RetainDataType.DataRealDrive;
	XINITRETAINDONE : BOOL;
	XNORETAINHANDLING : BOOL;
	PRETAINDATA : POINTER TO L_MC1P_uRetainData;
	XRETAINDATAAVAILABLE : BOOL;
	APOSDATA : ARRAY [0..3] OF L_MC1P_uRetainData;
	WIDXCNTPOSDATA : WORD;
	XINITRETAINBUFFER : BOOL;
	DWINITTIMER : DWORD;
	XSENDFRAMEATTASKSTART : BOOL;
	XDRIVELOADENCODER : BOOL;
	XDRIVELOADENCODEREVALUATECONFIG : BOOL;
	XDRIVELOADENCODERORIENTATION : BOOL;
	ALRHISTORYSETPOSITION : ARRAY [0..c_wMaxSetValueDelay] OF LREAL;
	ALRHISTORYSETPOSROUNDS : ARRAY [0..c_wMaxSetValueDelay] OF LREAL;
	WHISTORYIDX : WORD := 0;
	LRFEPOSDIFFPOSCONTROL : LREAL;
	XFESETPOSVALID : BOOL;
	DWFECOUNTER : DWORD;
	LRRESIDUALPOSFILTER : LREAL;
	LRRESIDUALVEL : LREAL;
	EQUICKSTOPOPTION : L_MC1P_QuickStopOption := L_MC1P_QuickStopOption.StayInQSP;
	ECONTROLMODEOLD : L_MC1P_ControlMode;
	XUSEIPMODENOTCSP : BOOL := FALSE;
	XUSEVLMODENOTCSV : BOOL := FALSE;
	XPDINEQPDOUT : BOOL;
	LWIDENTDRIVESWITCHOFF : LWORD := 0;
	WOFFSETDRIVEPARA : WORD := 0;
	WMCTRLMODEDRIVE : USINT := 1;
	XVFCMODE : BOOL := FALSE;
	XUSEEXTENCODERFORPOSCTRL : BOOL;
	ELSTCSFERRORID : L_IE1P_Error;
	LRSPEEDLIMITSLSINT : LREAL;
	XPOSRECONSTRUCTINEXTERNAL : BOOL := FALSE;
	XLINEARENCODER : BOOL := FALSE;
	LRMAXPOSITIONDIFF : LREAL := 0;
	XFORWARDECATSLAVEERROR : BOOL := TRUE;
	XIGNOREFOLLOWINGERRORRESET : BOOL := FALSE;
	LRSTAYINLASTSTATEOFFSETBRAKE : LREAL;
	XSTAYINLASTSTATEHANDLINGBRAKE : BOOL;
	XSTAYINLASTSTATEHANDLINGBRAKEOLD : BOOL;
	ADIACTPOSITION_INCR : ARRAY [0..15] OF DINT;
	EALLOWEDSERVICEDIRECTION : L_MC1P_ServiceDirection;
	WFDBSTATUSWORD : WORD;
	XENCODERSTATUSVALIDFORRETAINHANDLING : BOOL;
	XENCODERSTATUSVALIDFORRETAINHANDLINGOLD : BOOL;
	XRESTORERETAINPOSAFTERENCERROR : BOOL;
	XFIRSTSTORERETAINDONE : BOOL := FALSE;
	XRESETRETAINENCERRORAFTERMAINSWITCH : BOOL;
	USIHOMEPOSPERMANTENTSET : USINT;
	ITFAXISSIMULATION : L_MC1P_IAxisSimulationInterface;
	XAXISSIMULATIONACTIVE : BOOL;
	DWFIRSTOPTIMER : DWORD;
	DWPRODUCTCODE : DWORD;
	ITFCOMM : L_MC1P_ICommunication;
	ITFEXTENDEDMAPPINGACCESS : L_MC1P_IExtendedMappingAccess;
	M_PMASTERCONNECTOR : POINTER TO IoConfigConnector;
	XCHECKCOMMUNICATIONSTATE : BOOL := TRUE;
	M_PPDOINFOCONNECTOR : POINTER TO IoConfigConnector;
	XMOTIONUTISINTERNCONNECTED : BOOL := FALSE;
	CONNECTEDDRIVEUTILS : L_MC1P_IDriveUtils;
	ITFDRIVESCALING : L_MC1P_IDriveScaling;
	SCPARCMDAUTOTUNING : L_MC1P_AutotuningPara;
	ITFCMDAUTOTUNING : L_MC1P_IAxisCommmand_Autotuning;
	ITFCMDBRAKETEST : L_MC1P_IAxisCommmand;
	ITFCMDBRAKEGRINDIN : L_MC1P_IAxisCommmand;
	ITFDRIVESPECIFIC : L_MC1P_IDriveSpecificImplBase := DriveSpecificBasic;
	BRAKETESTCOMMAND : USINT;
	BRAKEGRINDINCOMMAND : USINT;
	SCPARBRAKE : L_MC1P_BrakePara;
	SCPARBRAKEGRINDIN : L_MC1P_BrakeCmdBrakeGrindInPara;
	SCPARBRAKETEST : L_MC1P_BrakeCmdBrakeTestPara;
	XTACIAADVANCED : BOOL;
	XQSPATFASTSTOP : BOOL;
	ITFGENERICIMPL : L_MC1P_IGenericAxisConfiguration;
	ITFFUNCTIONCONNECTION : L_IF1P_IFunctionConnection;
	ITFCONFIGDRIVE : L_MC1P_IConfigureDrive;
	ITFRETAINHANDLING : L_MC1P_IRetainHandling;
	ITFRETAINHANDLINGBASE : L_MC1P_IRetainHandling;
	UDRIVEDATA : L_MC1P_DriveSpecificContainer;
	FB_NODECONNCECTIONSTATUS : L_IF1P_Status;
	C_WMAXSETVALUEDELAY : WORD := 7;
	C_WMAXTRANSELEM : WORD := 20;
	C_WMAXRECELEM : WORD := 38;
	C_WMAXTRANSELEMADD : WORD := 5;
	C_WMAXRECELEMADD : WORD := 5;
	AXISSLOT : L_MC1P_AxisSlot;
	CIA402ADVANCEDAXIS : BOOL;
	DRIVESPECIFICBASIC : L_MC1P_IDriveSpecificImplBase;
	GETITFBRAKE : L_MC1P_IAXIS_REF_BRAKE;
	GETITFCMDBRAKEGRINDIN : L_MC1P_IAxisCommmand;
	GETITFCMDBRAKETEST : L_MC1P_IAxisCommmand;
	HOMEPOSPERMANTENTSETACTIVE : BOOL;
	HOMEPOSPERMANTENTSETACTIVELOADENCODER : BOOL;
	HOMESEQUENCESTATE : WORD;
	QSPATFASTSTOPEND : BOOL;
	RESETFOLLOWINGERRORATFASTSTOPEND : BOOL;
	SERVICEDIRECTION : L_MC1P_ServiceDirection;
END_VAR
END_FUNCTION_BLOCK

METHOD CALCACTPOSUNFILTERED : LREAL
END_METHOD

METHOD CALCACTVALUES
END_METHOD

METHOD CALCCONTOLLER
END_METHOD

METHOD CALCDRIVEHOMEOFFSET : DINT
VAR_INPUT
	LROLDPOS : LREAL;
	LRNEWPOSPOS : LREAL;
END_VAR
END_METHOD

METHOD CHECKFOLLOWINGERROR : BOOL
END_METHOD

METHOD CHECKPLNOTVALID : BOOL
END_METHOD

METHOD CHECKSETPOSINWINDOW : BOOL
END_METHOD

METHOD COMPENSATELOADPOSOFFSET
END_METHOD

METHOD CONVACTPOS : LREAL
VAR_INPUT
	LIPOS : LINT;
	LRRESIDUALPOS : LREAL;
END_VAR
VAR_OUTPUT
	LRROUNDS : LREAL;
END_VAR
END_METHOD

METHOD CORRECTHISTORY
VAR_INPUT
	LRPOSOFFSET : LREAL;
END_VAR
END_METHOD

METHOD ENABLEDRIVE : BOOL
VAR_INPUT
	XENABLE : BOOL;
END_VAR
END_METHOD

METHOD GENACTVALUES
END_METHOD

METHOD GETACTVEL : LREAL
END_METHOD

METHOD GETACTIVEPOSCTRLADAPTVALUE : LREAL
END_METHOD

METHOD GETACTIVEQUICKSTOPOPTION : L_MC1P_QuickStopOption
END_METHOD

METHOD GETBRAKE : POINTER TO L_MC1P_BrakeControlBase
END_METHOD

METHOD GETBRAKESERVICE : POINTER TO L_MC1P_BrakeService
END_METHOD

METHOD GETCAUSEOFCINH : WORD
END_METHOD

METHOD GETDRIVESTATE : BOOL
END_METHOD

METHOD GETPOINTERTOTPAXIS : POINTER TO _AXIS_REF_REAL
END_METHOD

METHOD GETREFERENCETORQUE : LREAL
END_METHOD

METHOD GETSTATUSWORDS
VAR_OUTPUT
	STATUSWORD1 : WORD;
	STATUSWORD2 : WORD;
	STATUSWORD3 : WORD;
	STATUSWORD4 : WORD;
END_VAR
END_METHOD

METHOD GETTPWITHPOSITIONACTIVE : BOOL
VAR_INPUT
	SITPNUMBER : SINT;
END_VAR
END_METHOD

METHOD GETTPWITHTIMESTAMPACTIVE : BOOL
VAR_INPUT
	SITPNUMBER : SINT;
END_VAR
END_METHOD

METHOD GETVELERRORLASTTASKCYCLES
VAR_IN_OUT
	ALRVELERR : ARRAY [0..3] OF LREAL;
END_VAR
END_METHOD

METHOD HOMECONFIG
VAR_INPUT
	PAXIS : POINTER TO _AXIS_REF_REAL;
	PPW : POINTER TO L_DCO_WriteDriveParameter;
	PHOMEDATA : POINTER TO L_MC1P_HomeParameter;
	LRPOSITION : LREAL;
	PWSTEP : POINTER TO WORD;
END_VAR
VAR_OUTPUT
	XDONE : BOOL;
	XERROR : BOOL;
END_VAR
END_METHOD

METHOD POSDIFFTOSPEEDINC : DINT
VAR_INPUT
	DIPOSDIFF : DINT := 0;
	DWFACTOR : DWORD := 1000;
END_VAR
END_METHOD

METHOD RESETACTPOS
END_METHOD

METHOD RESETCIACTRLWORD
END_METHOD

METHOD RESETERRORSTATEOFCOMMANDS : BOOL
END_METHOD

METHOD RESETFOLLOWINGERROR
END_METHOD

METHOD RESETHOMEPOS2
VAR_INPUT
	ERESETINFO : L_IE1P_Error;
END_VAR
END_METHOD

METHOD RESETHOMEPOSLOADENCODER
VAR_INPUT
	ERESETINFO : L_IE1P_Error;
END_VAR
END_METHOD

METHOD SERVICEMODEHANDLINGINDRIVEACTIVE : BOOL
END_METHOD

METHOD SETACTPOSITION
VAR_INPUT
	POSITION : LREAL;
	RELATIVE : BOOL;
END_VAR
END_METHOD

METHOD SETAXISSTATUSWORD
END_METHOD

METHOD SETCOMMANDINTERFACEAUTOTUNING
VAR_INPUT
	ITF : L_MC1P_IAxisCommmand_Autotuning;
END_VAR
END_METHOD

METHOD SETCONTROLWORDS
VAR_INPUT
	CONTROLWORD1 : WORD;
	CONTROLWORD2 : WORD;
	CONTROLWORD3 : WORD;
	CONTROLWORD4 : WORD;
END_VAR
END_METHOD

METHOD SETDCBRAKE
VAR_INPUT
	XSETDCBRAKE : BOOL;
END_VAR
VAR_OUTPUT
	XDCBRAKEACTIVE : BOOL;
END_VAR
END_METHOD

METHOD SETHOMEPOSITION2
VAR_INPUT
	POSITION : LREAL;
	RELATIVE : BOOL;
	XRESTARTPOSITIONING : BOOL := FALSE;
	EHOMEPOSINFO : L_IE1P_Error;
END_VAR
END_METHOD

METHOD SETINERTIAADAPT
VAR_INPUT
	LRADAPT : LREAL;
END_VAR
END_METHOD

METHOD SETPOSCTRLADAPTVALUE
VAR_INPUT
	LRADAPT : LREAL;
END_VAR
END_METHOD

METHOD SETSPEEDCTRLLOADVALUE
VAR_INPUT
	XLOAD : BOOL;
	LRVALUE : LREAL;
END_VAR
END_METHOD

METHOD SETVALFORCHECKFOLLOWINGERROR : BOOL
VAR_INPUT
	LRPOSDIFF : LREAL;
END_VAR
END_METHOD

METHOD SPEEDEQZERO : BOOL
VAR_INPUT
	LRSPEEDIN : LREAL;
END_VAR
END_METHOD

METHOD SPEEDTOPOSDIFFINC : DINT
VAR_INPUT
	DISPEED : DINT := 0;
	DWFACTOR : DWORD := 1000;
END_VAR
VAR_IN_OUT
	DIRES : DINT;
END_VAR
END_METHOD

METHOD CALLRECIEVEPARAMETER
END_METHOD

METHOD CALLTRANSMITPARAMETER
END_METHOD

METHOD CONFIGUREAXIS
END_METHOD

METHOD CONFIGUREAXIS2
END_METHOD

METHOD CONFIGUREAXISCONNECTOR
END_METHOD

METHOD CONNECTCMDITFAUTOTUNING
END_METHOD

METHOD FINISHDRIVECONFIG
END_METHOD

METHOD GETTRANSMITCYCLESACTSETPOS : LREAL
END_METHOD

METHOD REGISTERAXISPROPERTIES
END_METHOD

METHOD RESETDATA : BOOL
END_METHOD

METHOD SETAXISPROPERTIES
VAR_INPUT
	XUSEVIRTUAL : BOOL;
END_VAR
END_METHOD

METHOD SETBASICINITIALISATION
VAR_IN_OUT
	AXIS : _AXIS_REF_REAL;
END_VAR
END_METHOD

METHOD SETDRIVECONFIG
VAR_OUTPUT
	XDONE : BOOL;
	XERROR : BOOL;
	WERRORID : WORD;
END_VAR
END_METHOD

METHOD SETSPEEDCTRLLIMITATION : BOOL
VAR_INPUT
	XLIMIT : BOOL;
END_VAR
END_METHOD

METHOD CHECKAVAILABLECONTROLMODE : BOOL
END_METHOD

METHOD CONFIGURECONTROLMODE
VAR_OUTPUT
	EERRORID : L_IE1P_Error;
END_VAR
END_METHOD

METHOD GETDEFAULTCONTROLMODE : L_MC1P_ControlMode
END_METHOD

METHOD GETINTCONTROLMODE : SINT
VAR_INPUT
	ECONTROLMODE : L_MC1P_ControlMode;
END_VAR
END_METHOD

METHOD SELECTPOSITIONMODE
VAR_INPUT
	XPOSCTRLPLC : BOOL;
	XKEEPACTPOSPRIORFDB : BOOL := FALSE;
	XRESTARTPOSITIONING : BOOL := FALSE;
END_VAR
END_METHOD

METHOD SELECTSPEEDMODE
VAR_INPUT
	XKEEPACTPOSPRIORFDB : BOOL := FALSE;
	XRESTARTPOSITIONING : BOOL := FALSE;
END_VAR
END_METHOD

METHOD SELECTTORQUEMODE
END_METHOD

METHOD SETCONTROLMODE : BOOL
VAR_INPUT
	ECONTROLMODE : L_MC1P_ControlMode := L_MC1P_ControlMode.PosCtrlDrive;
	XKEEPACTPOSPRIORFDB : BOOL := FALSE;
	XRESTARTPOSITIONING : BOOL := FALSE;
END_VAR
VAR_OUTPUT
	EERRORID : L_IE1P_Error;
END_VAR
END_METHOD

METHOD SETCONTROLERITF
VAR_INPUT
	ITFCONTROLERNEW : L_MC1P_IControllerInterface;
END_VAR
END_METHOD

METHOD SWITCHPOSITIONFEEDBACK
VAR_INPUT
	XPOSFROMPLC : BOOL;
	XKEEPACTPOSPRIORFDB : BOOL := FALSE;
	XRESTARTPOSITIONING : BOOL := FALSE;
END_VAR
END_METHOD

METHOD CALCCYCLELENGTH
END_METHOD

METHOD CALCULATESCALING : BOOL
END_METHOD

METHOD CHECKVALIDPOSRESOLUTION : BOOL
VAR_INPUT
	DWPOSRESOLUTION : DWORD;
END_VAR
END_METHOD

METHOD GETVIRTUAL : BOOL
END_METHOD

METHOD MACHINEDATACHANGED : BOOL
END_METHOD

METHOD WRITENEWMACHINEDATA
VAR_INPUT
	LRFEEDCONSTANTNEW : LREAL := 360.0;
	DWGEARDENOMINATORNEW : DWORD := 1;
	DWGEARNUMERATORNEW : DWORD := 1;
	DWADDGEARDENOMINATORNEW : DWORD := 1;
	DWADDGEARNUMERATORNEW : DWORD := 1;
	DWPOSRESOLUTIONNEW : DWORD := 65536;
	XORIENTATIONNEW : BOOL := FALSE;
	ETRAVERSINGRANGENEW : L_MC1P_TraversingRange := L_MC1P_TraversingRange.Limited;
	LRCYCLELENGTHNEW : LREAL := 360.0;
END_VAR
END_METHOD

METHOD CALCSCALEFUNCTIONS
VAR_INPUT
	OFFSET : DWORD;
	INDEX : WORD;
END_VAR
END_METHOD

METHOD SETCONTROLMODEPARAMETER
END_METHOD

METHOD SETPOSCONTROLPARAMETER
END_METHOD

METHOD GENLOGENTRY : BOOL
VAR_INPUT
	PPOSDATA : POINTER TO L_MC1P_uRetainData;
END_VAR
END_METHOD

METHOD GENERATEENCODERSTATUSFORRETAINHANDLING : BOOL
VAR_INPUT
	WFDBSTATUSWORD : WORD;
END_VAR
END_METHOD

METHOD RESETRETAINHANDLING : BOOL
END_METHOD

METHOD RESTOREACTPOS
VAR_INPUT
	PPOSDATA : POINTER TO L_MC1P_uRetainData;
END_VAR
END_METHOD

METHOD RESTOREACTPOSBASE
VAR_INPUT
	PPOSDATA : POINTER TO L_MC1P_uRetainData;
END_VAR
END_METHOD

METHOD RESTOREADDITIONALRETAINDATA
VAR_INPUT
	PDATA : POINTER TO L_MC1P_uRetainData;
END_VAR
END_METHOD

METHOD RETAINHANDLING : BOOL
END_METHOD

METHOD STOREACTPOS
VAR_INPUT
	PPOSDATA : POINTER TO L_MC1P_uRetainData;
END_VAR
END_METHOD

METHOD STOREADDITIONALRETAINDATA
VAR_INPUT
	PDATA : POINTER TO L_MC1P_uRetainData;
END_VAR
END_METHOD

METHOD STOREDATA
VAR_INPUT
	PDATA : POINTER TO DWORD;
END_VAR
END_METHOD

METHOD CALCOPTIMIZEDMAPPINGINFO : BOOL
END_METHOD

METHOD GETRECEIVEDATA : DWORD
VAR_INPUT
	LWMASK : LWORD;
END_VAR
END_METHOD

METHOD GETRECEIVEDATAIMPL : DWORD
VAR_INPUT
	LWMASK : LWORD;
END_VAR
END_METHOD

METHOD GETTRANSMITDATA : DWORD
VAR_INPUT
	LWMASK : LWORD;
END_VAR
END_METHOD

METHOD GETTRANSMITDATAIMPL : DWORD
VAR_INPUT
	LWMASK : LWORD;
END_VAR
END_METHOD

METHOD GETTRANSMITDATALREAL : LREAL
VAR_INPUT
	LWMASK : LWORD;
END_VAR
END_METHOD

METHOD GETTRANSMITDATALREALIMPL : LREAL
VAR_INPUT
	LWMASK : LWORD;
END_VAR
END_METHOD

METHOD RECEIVEPARAMETER
VAR_INPUT
	WPARAMETER : WORD;
	PADRESS : POINTER TO BYTE;
	WSIZE : WORD;
END_VAR
END_METHOD

METHOD RECEIVEPARAMETERCALC
VAR_IN_OUT
	DATA : ARRAY [1..L_MC1P_Constants.gc_Rec_MaxDataIndex] OF POINTER TO L_MC1P_MappedElement;
END_VAR
END_METHOD

METHOD TRANSMITPARAMETER
VAR_INPUT
	WPARAMETER : WORD;
	PADRESS : POINTER TO BYTE;
	WSIZE : WORD;
END_VAR
END_METHOD

METHOD TRANSMITPARAMETERCALC
VAR_IN_OUT
	DATA : ARRAY [1..L_MC1P_Constants.gc_Trans_MaxDataIndex] OF POINTER TO L_MC1P_MappedElement;
END_VAR
END_METHOD

METHOD PDCONVACTPOS : DINT
VAR_INPUT
	DIINPUT : DINT;
END_VAR
END_METHOD

METHOD PDCONVACTVEL : DINT
VAR_INPUT
	DIINPUT : DINT;
END_VAR
END_METHOD

METHOD PDCONVSETPOS : DINT
VAR_INPUT
	XSETEQACTONDISABLED : BOOL;
END_VAR
END_METHOD

METHOD PDCONVSPEEDCTRLINT : INT
VAR_INPUT
	LRINPUT : LREAL;
END_VAR
END_METHOD

METHOD PDCONVTPPOS : DINT
VAR_INPUT
	DIPOS : DINT;
END_VAR
END_METHOD

METHOD CALLSIMULATION
VAR_INPUT
	CALLSTATE : L_UBUP_StateHandleCase;
END_VAR
END_METHOD

METHOD SETAXISSIMULATION : BOOL
VAR_INPUT
	ITFAXISSIMULATION : L_MC1P_IAxisSimulationInterface;
END_VAR
END_METHOD

METHOD CALCAFTERREADINPUTS : INT
END_METHOD

METHOD CALCBEFOREREADINPUTS : INT
END_METHOD

METHOD CALCBEFOREWRITEOUTPUTS : INT
END_METHOD

METHOD GETIECADRESS
END_METHOD

METHOD INITIALIZE : UDINT
VAR_INPUT
	WMODULETYPE : UINT;
	DWINSTANCE : UDINT;
	PCONNECTOR : POINTER TO IoConfigConnector;
END_VAR
END_METHOD

METHOD IODRVREADPARAMETER : UDINT
VAR_INPUT
	PCONNECTOR : POINTER TO IoConfigConnector;
	PPARAMETER : POINTER TO IoConfigParameter;
	PDATA : POINTER TO BYTE;
	DWBITSIZE : DWORD;
	DWBITOFFSET : DWORD;
END_VAR
END_METHOD

METHOD ISINCLUDEDINRECEIVEDATA : BOOL
VAR_INPUT
	LWMASK : LWORD;
END_VAR
END_METHOD

METHOD ISINCLUDEDINTRANSMITDATA : BOOL
VAR_INPUT
	LWMASK : LWORD;
END_VAR
END_METHOD

METHOD FB_INIT : BOOL
VAR_INPUT
	BINITRETAINS : BOOL;
	BINCOPYCODE : BOOL;
END_VAR
END_METHOD

METHOD GETMAGNETISATIONFINISHED : BOOL
END_METHOD

METHOD CONNECTMOTIONUTILS
VAR_INPUT
	DRIVEUTILS : L_MC1P_IDriveUtils;
	AXISEXTENSION : L_MC1P_IAxisExtension;
END_VAR
END_METHOD

METHOD CONNECTMOTIONUTILSFORINTERNALUSE : BOOL
VAR_INPUT
	DRIVEUTILS : L_MC1P_IDriveUtils;
	AXISEXTENSION : L_MC1P_IAxisExtension;
	ITFRETAIN : L_MC1P_IRetainHandling;
END_VAR
END_METHOD

METHOD DISCONNECTMOTIONUTILS : BOOL
VAR_INPUT
	EDISCONNECTMODE : L_IF1P_DisconnectMode;
END_VAR
END_METHOD

METHOD FINDANDCONNECTMOTIONUTILS
END_METHOD

(* ---- _AXIS_REF_UNIVERSAL.pou ---- *)
FUNCTION_BLOCK _AXIS_REF_UNIVERSAL EXTENDS _AXIS_REF_COM
VAR
	FBDRIVESPECIFIC : L_MC1P_DriveSpecific_Basic;
	AXISEXTENSIONFACTORY : L_MC1P_UniversalAxisFactory;
	ITFDRIVEUTILSTOCONNECT : POINTER TO L_MC1P_IDriveUtils;
	ITFAXISEXTENSION : L_MC1P_IAxisExtension;
	RETAINMANAGEMENT : L_MC1P_MotionUtilsRetainHandlingUniversal;
	UITYPE : UINT := 1;
	DRIVESPECIFICBASIC : L_MC1P_IDriveSpecificImplBase;
END_VAR
END_FUNCTION_BLOCK

METHOD CALCAFTERREADINPUTS : INT
END_METHOD

METHOD CONNECTASYNC : BOOL
END_METHOD

METHOD CREATEAXISEXTENSION : L_MC1P_IAxisExtension
VAR_INPUT
	EAXISEXTENSIONTYPE : L_MC1P_AxisExtensionTypes;
END_VAR
END_METHOD

METHOD FINDANDCONNECTMOTIONUTILS
END_METHOD

METHOD FINDDRIVEUTILSINMOTIONCONNECTOR : BOOL
VAR_INPUT
	PECATSLAVECONNECTOR : POINTER TO IoConfigConnector;
	SUBDEVICE : UINT;
END_VAR
END_METHOD

METHOD INITIALIZE : UDINT
VAR_INPUT
	WMODULETYPE : UINT;
	DWINSTANCE : UDINT;
	PCONNECTOR : POINTER TO IoConfigConnector;
END_VAR
END_METHOD

METHOD SETGENERICCONFIGURATION
VAR_INPUT
	ITFGENERICCONFIG : L_MC1P_IGenericAxisConfiguration;
END_VAR
END_METHOD

METHOD FB_INIT : BOOL
VAR_INPUT
	BINITRETAINS : BOOL;
	BINCOPYCODE : BOOL;
END_VAR
END_METHOD

METHOD CONNECTDEVICE : UINT
VAR_INPUT
	DEVICEMODULEHANDLER : L_IMHP_IModuleHandler;
	UISUBDEVICE : UINT := 0;
	EDISCONNECTMODE : L_IF1P_DisconnectMode;
	XDISCONNECTEXISTINGCONNECTION : BOOL;
END_VAR
VAR_OUTPUT
	ITFCONNECTIONFBSTATUS : L_IF1P_IStatus;
END_VAR
END_METHOD

METHOD DISCONNECTDEVICE : UINT
VAR_INPUT
	EDISCONNECTMODE : L_IF1P_DisconnectMode;
	XBUSYBEFORE : BOOL;
END_VAR
VAR_OUTPUT
	ITFCONNECTIONFBSTATUS : L_IF1P_IStatus;
END_VAR
END_METHOD

METHOD GEFUNCTIONTINSTANCEPOINTER : POINTER TO BYTE
END_METHOD

METHOD GETCONNECTEDDEVICE : L_IMHP_IModuleHandler
VAR_OUTPUT
	UISUBDEVICE : UINT := 0;
	XVALID : BOOL;
	ITFCONNECTIONFBSTATUS : L_IF1P_IStatus;
END_VAR
END_METHOD

METHOD GETCONNECTIONDIAGNOSTIC
VAR_OUTPUT
	WUSEDBY_COMP : WORD;
	WUSEDBY_SUBCOMP : WORD;
	WACTIVEMODE : WORD;
	WSUBDEVICE : WORD;
	SCONNECTIONSOURE : STRING;
END_VAR
END_METHOD

METHOD GETITFCONNECTSTATUS
VAR_OUTPUT
	ITFCONNECTIONFBSTATUS : L_IF1P_IStatus;
END_VAR
END_METHOD

(* ---- _AXIS_REF_VMA.pou ---- *)
FUNCTION_BLOCK _AXIS_REF_VMA EXTENDS AXIS_REF
VAR_OUTPUT
	LRSETPOSITIONEFFECTIVE : LREAL;
	LRSETVELOCITYEFFECTIVE : LREAL;
	LRSETACCELERATIONEFFECTIVE : LREAL;
END_VAR
VAR
	LRACSSETVALUEFILTERPOSDEVIATION : LREAL;
END_VAR
END_FUNCTION_BLOCK

METHOD ADDTRACKINGOFFSET
VAR_INPUT
	LRPOSOFFSET : LREAL;
	LRVELOFFSET : LREAL;
	LRACCOFFSET : LREAL;
END_VAR
END_METHOD

METHOD ERRORSTOP
END_METHOD

METHOD GENACTVALUES
END_METHOD

METHOD PASSTHROUGHTRACKINGOFFSETRESET
VAR_INPUT
	LRDISTANCE : LREAL;
END_VAR
END_METHOD

METHOD SETACSFILTERDEVIATION
VAR_INPUT
	LRACSFILTERPOSDEVIATION : LREAL;
END_VAR
END_METHOD

METHOD SETACTVALUES
VAR_INPUT
	LRACTPOS : LREAL;
	TASKCYCLETIME : LREAL;
END_VAR
END_METHOD

METHOD CONFIGUREAXISCONNECTOR
END_METHOD

METHOD REGISTERAXISPROPERTIES
END_METHOD

METHOD UPDATEFATHERCONNECTOR
END_METHOD

METHOD CALCBEFOREWRITEOUTPUTS : INT
END_METHOD

METHOD INITIALIZE : UDINT
VAR_INPUT
	WMODULETYPE : UINT;
	DWINSTANCE : UDINT;
	PCONNECTOR : POINTER TO IoConfigConnector;
END_VAR
END_METHOD

METHOD QUERYINTERFACE : POINTER TO POINTER TO BYTE
VAR_INPUT
	IID : DWORD;
	PRESULT : POINTER TO UDINT;
END_VAR
END_METHOD

METHOD FB_INIT : BOOL
VAR_INPUT
	BINITRETAINS : BOOL;
	BINCOPYCODE : BOOL;
END_VAR
END_METHOD

(* ---- _L_MC1P_ANALOGINPUTSPEEDCTRL.pou ---- *)
FUNCTION_BLOCK _L_MC1P_ANALOGINPUTSPEEDCTRL
VAR_INPUT
	WINPUT : WORD;
	WUPPERLIM : WORD := 10000;
	WLOWERLIM : WORD := 0;
	LRUPPERSPEEDLIM : LREAL := 1000;
	LRLOWERSPEEDLIM : LREAL := 0;
	LRDEADBAND : LREAL := 5;
	LRFILTTIME : LREAL := 0.01;
	LRACC : LREAL := 1000;
	LRDEC : LREAL := 1000;
	LRJERK : LREAL := 100000;
	XNEGATIVEDIRECTION : BOOL;
END_VAR
VAR_OUTPUT
	LRSETSPEEDOUT : LREAL;
END_VAR
VAR
	LRINPUTSCALED : LREAL;
	LRSPEEDSETPOINT : LREAL;
	L_D94A_FILTER : L_USPP.L_USPP_PT1Filter;
	L_MC1P_RAMPGENERATOR1 : L_MC1P_RampGenerator;
END_VAR
END_FUNCTION_BLOCK

(* ---- AXIS_REF.pou ---- *)
FUNCTION_BLOCK AXIS_REF EXTENDS L_DCO_AXIS_REF_BASE
VAR_INPUT
	LRVELOVERRIDE : LREAL := 1.0;
	LRACCOVERRIDE : LREAL := 1.0;
	LRJERKOVERRIDE : LREAL := 1.0;
	LRCOMMANDEDPOSITION : LREAL;
	LRCOMMANDEDVELOCITY : LREAL;
	LRCOMMANDEDACCELERATION : LREAL;
	LRSETVELOCITYLIMITHIGH : LREAL := 0;
	LRSETVELOCITYLIMITLOW : LREAL := 0;
	LRTORQUELIMHIGH : LREAL;
	LRTORQUELIMLOW : LREAL;
	LRTORQUELIMAUX : LREAL;
	SITORQUELIMDIR : SINT;
	XDELETETORQUELIM : BOOL;
	XSETTORQUELIMAUX : BOOL;
	XTORQUELIMHIGHFROMAPP : BOOL;
	XTORQUELIMLOWFROMAPP : BOOL;
	ITORQUELIMHIGHPCT : INT := 2000;
	ITORQUELIMLOWPCT : INT := 2000;
	EDIRECTION : MC_DIRECTION;
	XDRIVEENABLE : BOOL;
	XERRORRESET : BOOL;
	LRREFOFFSET : LREAL;
	LRREFOFFSETACT : LREAL;
	XENABLEPOSITIVE : BOOL := TRUE;
	XENABLENEGATIVE : BOOL := TRUE;
	LRSETSUPERACC : LREAL;
	LRSETSUPERVEL : LREAL;
	LRSETSUPERPOS : LREAL;
	LRSETMOVEACC : LREAL;
	LRSETMOVEVEL : LREAL;
	LRSETMOVEPOS : LREAL;
	XBUFCMDDONE : BOOL;
	XBUFRESTART : BOOL;
	LRPROFILESPEEDFIRST : LREAL;
	LRPROFILETARGETSPEED : LREAL;
	DWBUFFERCMD : __XWORD;
	XDISABLEERRORLOGGING : BOOL;
	XMOVEFUNBUSY : BOOL;
	XSUPERFUNBUSY : BOOL;
	LRCOMMANDEDPOSABSOLUT : LREAL;
	XRESETFOLLOWINGERROR : BOOL;
	XSETAXISQSP : BOOL;
	XSETDRIVEQSP : BOOL;
	EAXISSTATE : L_MC1P_AXIS_STATE := 2;
	LRSETPOSITION : LREAL := 0.0;
	LRSETVELOCITY : LREAL := 0.0;
	LRSETACCELERATION : LREAL := 0.0;
	LRSETTORQUE : LREAL := 0.0;
	LRVLTARGETVEL : LREAL := 0.0;
	LRLIMITEDVELOCITY : ARRAY [1..4] OF LREAL;
	LRLIMITEDDECTIME : ARRAY [1..4] OF LREAL;
	LRRESETSLSOFFSETVELOCITY : LREAL;
	DWLIMITERCONTROLACT : DWORD;
	SCSTOPAXISBYAPPL : L_MC1P_StopOperation;
	XSTAYINLASTSTATEREQUEST : BOOL;
	XMOVELASTSETPOSREQUEST : BOOL;
	LRSETVELMOVELASTSETPOS : LREAL;
	LRSETACCMOVELASTSETPOS : LREAL;
	LRSETDECMOVELASTSETPOS : LREAL;
	LRSETJERKMOVELASTSETPOS : LREAL;
	EDIRECTIONMOVELASTSETPOS : MC_DIRECTION;
	EDIRECTIONACTPROFILE : MC_DIRECTION;
	WAXISCONTROL : WORD := 0;
	XALLOWCHANGEOFCINHPAR : BOOL := FALSE;
	LRMOVEVELOFFSETVEL : LREAL;
	EOPTIMIZEDPROFILECALCULATIONMODE : UINT := 1;
	XLEAVESERVICESTATE : BOOL;
	XLEAVESERVICESTATEDISABLEDRIVE : BOOL;
	WLEAVESERVICESTATEPOWID : WORD;
END_VAR
VAR_OUTPUT
	EDEVICE : L_MC1P_DriveType := 0;
	WAXISSTATUS : DWORD := 0;
	EACTIVEERRORID : WORD := 0;
	LRACTPOSITION : LREAL := 0.0;
	LRACTVELOCITY : LREAL := 0.0;
	LRACTACCELERATION : LREAL := 0.0;
	LRACTTORQUE : LREAL := 0.0;
	LRSETTORQUETODRIVE : LREAL := 0;
	LRACTFOLLOWINGERROR : LREAL := 0.0;
	LRMAXFOLLOWINGERROR : LREAL := 0.0;
	XVIRTUAL : BOOL;
	XAXISAVAILABLE : BOOL;
	EACTDIRECTION : MC_DIRECTION;
	LRDIRECTIONHYSTERESISPOS : LREAL;
	LRDIRECTIONHYSTERESISTOL : LREAL := 1E-06;
	XDRIVEENABLED : BOOL;
	XERROR : BOOL;
	XWARNING : BOOL;
	XDRIVEERROR : BOOL;
	XDRIVEWARNING : BOOL;
	DWDRIVEERRORID : DWORD;
	XHOMEPOSAVAILABLE : BOOL;
	XSWLIMITENABLED : BOOL;
	XSWLIMITPOS : BOOL;
	XSWLIMITNEG : BOOL;
	XHWLIMITPOS : BOOL;
	XHWLIMITNEG : BOOL;
	XSPEEDEQZERO : BOOL;
	XINPOSITION : BOOL;
	LRTASKCYCLE : LREAL := 0.001;
	LRINVTASKCYCLE : LREAL := 1000.0;
	LRSWLIMITPOS : LREAL := 0.0;
	LRSWLIMITNEG : LREAL := 0.0;
	LRLASTSETPOSITION : LREAL;
	LRLASTTARGETPOSITION : LREAL;
	XSTANDSTILLSETVELOCITY : BOOL;
	XSTANDSTILLACTVELOCITY : BOOL;
	XSTOACTIVE : BOOL;
	XVOLTAGEENABLED : BOOL;
	XAXISREADYTOSWITCHON : BOOL;
	XAXISREADYFORMOTION : BOOL;
	SCPAR : L_MC1P_ParAccess;
END_VAR
VAR
	DWAXISCONFIGSETTINGS : DWORD;
	XSETVALUESAVAILABLE : BOOL;
	BYSETVALUESVALID : BYTE;
	DWTASKYCLE_US : DWORD := 1000;
	XSUSPENDFOLLOWINGERRORINT : BOOL;
	XSUSPENDFOLLOWINGERROREXT : BOOL;
	LRMAXVELOCITYAPPLOLD : LREAL;
	LRMAXACCELERATIONAPPLOLD : LREAL;
	LRMAXJERKAPPLOLD : LREAL;
	LRSWLIMITPOSOLD : LREAL;
	LRSWLIMITNEGOLD : LREAL;
	XENABLEPOSOLD : BOOL;
	XENABLENEGOLD : BOOL;
	DWLIMITERCONTROLOLD : DWORD;
	LRLIMITEDVELOCITYOLD : ARRAY [1..4] OF LREAL;
	LRLIMITEDDECTIMEOLD : ARRAY [1..4] OF LREAL;
	LRLIMITEDJERKOLD : ARRAY [1..4] OF LREAL;
	ELIMITERSTOPREACTION : L_IE1P_SeverityLevel := L_IE1P_SeverityLevel.WARNING;
	XSWLIMITDISABLE : BOOL := FALSE;
	XSWLIMITPOSNEU : BOOL;
	XSWLIMITPOSISTAN : BOOL;
	XSWLIMITNEGNEU : BOOL;
	XSWLIMITNEGISTAN : BOOL;
	PBYCOUPLEDMASTERAXIS : POINTER TO BYTE;
	PBYCOUPLEDPHASINGMASTERAXIS : POINTER TO BYTE;
	LRPHASESHIFTPOS : LREAL;
	LRPHASESHIFTVEL : LREAL;
	LRPHASESHIFTACC : LREAL;
	LRPHASESHIFTPOSOLD : LREAL;
	LRPHASESHIFTVELOLD : LREAL;
	LRPHASESHIFTACCOLD : LREAL;
	XSETPHASESHIFTVALUES : BOOL;
	ETRAVERSINGRANGEACT : L_MC1P_TraversingRange := 0;
	LRCYCLELENGTHACT : LREAL := 360.0;
	XENABLEHWLIMITPOS : BOOL := TRUE;
	XENABLEHWLIMITNEG : BOOL := TRUE;
	XHWSIGNALNEG : BOOL := FALSE;
	XHWSIGNALPOS : BOOL := FALSE;
	BHWENSCHPOSNEU : BOOL := TRUE;
	BNOTIFYERRORHWLIMITPOSISTAN : BOOL;
	BHWENSCHNEGNEU : BOOL := TRUE;
	BNOTIFYERRORHWLIMITNEGISTAN : BOOL;
	XAXISISHOMESOURCE : BOOL;
	XHOMEPOSAVAILABLEDRIVE : BOOL;
	SCHOMEPARAMETER : L_MC1P_HomeParameter;
	LRHOMEPOSITION : LREAL;
	XPOSCTRL : BOOL;
	XTPSUPPORTED : BOOL := FALSE;
	XTPWITHTIMESTAMP : BOOL := FALSE;
	SNTPMAXCHANNEL : SINT;
	PG : L_MC1P_PosProfiler := STRUCT(wCalcProfileMode := 1);
	ITFPG_MOVEACTIVE : L_MC1P_IPosProfilerActive;
	PG_MOVE : L_MC1P_PosProfiler := STRUCT(wCalcProfileMode := 1);
	ITFPG_SUPERACTIVE : L_MC1P_IPosProfilerActive;
	PG_SUPER : L_MC1P_PosProfiler := STRUCT(wCalcProfileMode := 1);
	PG_DUMMY : L_MC1P_PosProfiler := STRUCT(wCalcProfileMode := 1);
	SCPARAMSTOP : L_MC1P_ProfileParameter;
	XCTRLMODECHANGEREQ : BOOL;
	LRCTRLMODECHANGEREQACTVEL : LREAL;
	PFBMOVEBASIC : POINTER TO L_MC1P_MoveBasic;
	PFBMOVEBASICSUPER : POINTER TO L_MC1P_MoveBasic;
	XRESTARTPOSITIONING : BOOL;
	LRSETPOSITIONOLD : LREAL;
	LRSETVELOCITYOLD : LREAL;
	LRSETACCELERATIONOLD : LREAL;
	WACTFUNID : WORD := 0;
	WACTSUPERFUNID : WORD := 0;
	WACTPHASEFUNID : WORD := 0;
	PSERRORINST : POINTER TO STRING;
	SERRORINST : STRING;
	ERRORMANAGER : L_IE1P_ErrorManager;
	ERRORRESETOCCUREDTIMEWITHOUTLEM : SYSTIME;
	ASCERRORINFO : REFERENCE TO ARRAY [0..7] OF L_IE1P_ErrorInformation;
	ASCWARNINGINFO : REFERENCE TO ARRAY [0..7] OF L_IE1P_ErrorInformation;
	WINITSTATE : WORD;
	PAPPLICATION : POINTER TO APPLICATION;
	ATPDATA : ARRAY [1..4] OF L_MC1P_TPData;
	ATPDATASAVE : L_MC1P_TPData;
	XHOMINGSUPPORTED : BOOL;
	EAXISSTATEOLD : L_MC1P_AXIS_STATE := L_MC1P_AXIS_STATE.Disabled;
	ECONTROLMODE : L_MC1P_ControlMode := L_MC1P_ControlMode.PosCtrlDrive;
	ECONTROLMODEDEFAULT : L_MC1P_ControlMode := L_MC1P_ControlMode.PosCtrlDrive;
	ECONTROLMODEDEFAULTINT : L_MC1P_ControlMode := L_MC1P_ControlMode.PosCtrlDrive;
	POSCTRLDRIVEAVAILABLE : L_IE1P_Error;
	POSCTRLPLCAVAILABLE : L_IE1P_Error;
	SPEEDCTRLDRIVEAVAILABLE : L_IE1P_Error;
	TORQUECTRLDRIVE : L_IE1P_Error;
	XDRIVEENABLEOLD : BOOL;
	XLOCKEDFORSINGLEMOTION : BOOL := FALSE;
	XHOMEABSSWITCH : BOOL;
	XHOMEABSSWITCHOVERWRITEACTIVE : BOOL;
	XRAMPTOSTANDSTILL : BOOL;
	XRAMPTOSTANDSTILLDONE : BOOL;
	XRAMPTOSTANDSTILLACTIVE : BOOL;
	XDRIVEENABLEDOLD : BOOL;
	XDRIVEENABLEDREAL : BOOL;
	XDRIVEENABLEDREALOLD : BOOL;
	LRFOLLOWINGERRORINT : LREAL;
	XSUPPORTBRAKE : BOOL := FALSE;
	XSUPPORTDCBRAKE : BOOL := FALSE;
	XUSEASVIRTUALEXT : BOOL := FALSE;
	XUSEASVIRTUALEXTACT : BOOL := FALSE;
	LRSETSUPERACCOLD : LREAL;
	LRSETSUPERVELOLD : LREAL;
	LRSETSUPERPOSOLD : LREAL;
	ITFPARA : L_MC1P_IPara;
	XFASTSTOPDONE : BOOL;
	XFASTSTOPDONESAVE : BOOL;
	XSETFASTSTOPINT : BOOL;
	XERRRORSTOPACTIVE : BOOL;
	XERRRORSTOPDONE : BOOL;
	XSETAXISQSPACTIVE : BOOL;
	XRAMPQSPSTARTCALLEDFROMAPP : BOOL;
	XDRIVEQSPACTIVE : BOOL;
	XDRIVEQSPACTIVEOLD : BOOL;
	XDRIVEQSPSET : BOOL;
	XSETDRIVEFAILQSP : BOOL;
	XSETDRIVEFAILCINH : BOOL;
	XDRIVEQSPDONE : BOOL;
	XDRIVEQSPDONESAVE : BOOL;
	ESTOPTYPE : WORD;
	POW : L_MC1P_Power_Internal;
	XOBERVERESWITCHONTIME : BOOL := TRUE;
	FBBASE : L_MC1P_Template_ForAxis;
	ABC : L_MC1P_AxisBasicControl_Internal;
	ABCDATA : L_MC1P_AxisBasicControlInstanceData;
	ITFENCODER : L_MC1P_IEncoderInterface;
	ITFENCODERHANDLER : L_MC1P_IEncoderInterface;
	LRSETTORQUEFROMAXESGROUP : LREAL := 0;
	EPRECONTROLMODE : L_MC1P_PreControlMode := L_MC1P_PreControlMode.Automatic;
	GUID : L_MC1P_AxisGUID;
	LRTORQUEPRECTRL : LREAL;
	LRTORQUESET : LREAL;
	XMOVEFUNBUSYOLD : BOOL;
	XMOVEFUNBUSYOLDOLD : BOOL;
	DWIODRVDEVICEID : DWORD;
	WIODRVDEVICETYPE : WORD;
	EDEVICEORIGIN : L_MC1P_DriveType := L_MC1P_DriveType.Virtual;
	EDEVICECLASS : L_MC1P_DeviceClass := L_MC1P_DeviceClass.VirtualAxis;
	DWTARGETID : DWORD := 0;
	XCTRLFIRMWARECHECKPASSED : BOOL := FALSE;
	XENABLELOGENTRY : BOOL := 1;
	ETRAVERSINGRANGE : L_MC1P_TraversingRange := 1;
	LRCYCLELENGTH : LREAL := 360.0;
	LRINVCYCLELENGTH : LREAL := (1.0 / 360.0);
	LRDEFAULTVELOCITY : LREAL := 0.0;
	LRDEFAULTACCELERATION : LREAL := 0.0;
	LRDEFAULTJERK : LREAL := 0.0;
	LRMAXVELOCITYAPPL : LREAL := 0.0;
	LRMAXACCELERATIONAPPL : LREAL := 0.0;
	LRMAXJERKAPPL : LREAL := 0.0;
	XENABLESWLIMIT : BOOL := 0;
	WBEHAVEONSWLIMIT : WORD := 1;
	LRDECERRORSTOP : LREAL := 3600.0;
	LRJERKERRORSTOP : LREAL := 0.0;
	XREAKTONMCFBERROR : BOOL := 1;
	LRWINDOWSTANDSTILL : LREAL := 0.0;
	LRWINDOWVELOCITYCONST : LREAL := 0.0;
	LRWINDOWTARGETREACHED : LREAL := 0.0;
	LRWINDOWTARGETREACHEDTIME : LREAL := 0.0;
	LRMODPOSTOLERANCE : LREAL := 0.0;
	XSETVALUEMONITORING : BOOL := 0;
	EPARAMETERINDEX : WORD := 101;
	DWPARABASEINDEX : DWORD;
	PPARA2 : L_SSYP.L_SSYP_EVTPARAM_CmpLenzeIPCSystemSoftPLCParaChanged;
	HEVENTPARWRITE : SysTypes.RTS_IEC_HANDLE;
	HINTERFACEPARWRITE : SysTypes.RTS_IEC_HANDLE;
	HEVENTDOWNLOADDONE : SysTypes.RTS_IEC_HANDLE;
	HINTERFACEDOWNLOADDONE : SysTypes.RTS_IEC_HANDLE;
	HEVENTRESETDONE : SysTypes.RTS_IEC_HANDLE;
	HINTERFACERESETDONE : SysTypes.RTS_IEC_HANDLE;
	ITFCALLBACK : CmpEventMgr.ICmpEventCallback;
	DWEVENTCOUNTER : DWORD;
	WENABLEDRIVEBLOCKEDBYOBJECTTRANSFER : WORD := 0;
	XUSEDBYAXESGROUP : BOOL;
	PUSEDAXESGROUP : POINTER TO BYTE;
	DWEVTINITCOUNT : DWORD;
	XNEWHOMEPOSLOADED : BOOL;
	DWSETPOSITIONCALLCYCLE : DWORD;
	XSETPOSITIONCALLCYCLEVALID : BOOL;
	AITFFILTER : ARRAY [1..c_MaxFilterInt] OF L_MC1P_ISetvalueManipulationInterface;
	XENABLEFILTER : BOOL;
	XFILTERAVAILABLE : BOOL;
	XIGNORFILTERINSTOP : BOOL := TRUE;
	XIGNORFILTERINSTOPITF : BOOL;
	XUSEFILTERVALUESFORSYNC : BOOL := FALSE;
	LRSETPOSITIONFILT : LREAL;
	LRSETVELOCITYFILT : LREAL;
	LRSETACCELERATIONFILT : LREAL;
	LRSETTORQUEFILT : LREAL;
	LRSETVALUEFILTERPOSDEVIATION : LREAL;
	XINTARGETSETVALUEFILTER : BOOL;
	XSUSPENDSETVALUEFILTERCALL : BOOL := FALSE;
	LRSETPOSITIONFILTOLD : LREAL;
	LRSETVELOCITYFILTOLD : LREAL;
	LRSETACCELERATIONFILTOLD : LREAL;
	LRSETTORQUEFILTOLD : LREAL;
	LRSETPOSROUNDSFILTOLD : LREAL;
	AITFCOMPENSATION : ARRAY [1..c_MaxFilterInt] OF L_MC1P_ICompensationInterface;
	LRCOMPENSATIONOFFSETPOS : LREAL;
	LRCOMPENSATIONOFFSETVEL : LREAL;
	LRCOMPENSATIONOFFSETACC : LREAL;
	LRACTPOSITIONUNFILTERED : LREAL;
	LRINTARGETPOS : LREAL;
	LRACTTIMETARGETREACHED : LREAL;
	XSETVALUEINTARGET : BOOL;
	XUSEACYCLIC : BOOL := FALSE;
	XFORCEACYCLICMODE : BOOL := FALSE;
	WAXISMODE : WORD := 1;
	WAXISMODEOLD : WORD := 255;
	LRTRANSMITCYCLESACTPOS : LREAL := 0.0;
	LRTRANSMITCYCLESSETPOS : LREAL := 1.0;
	XCONNECTORDISABLEDBYPROJECT : BOOL;
	XCONNECTORDISABLED : BOOL;
	XAXISDETECTIONBUSY : BOOL;
	XAXISDETECTED : BOOL;
	XCONFIGDONE : BOOL;
	XBASICINIT : BOOL := TRUE;
	XAXISCONNECTBUSY : BOOL;
	XAXISCONNECTDONE : BOOL;
	XPDOINTERFACEDISABLED : BOOL;
	XDRIVETESTMODEACTIVE : BOOL;
	LRACTPOSROUNDS : LREAL;
	LRSETPOSROUNDS : LREAL;
	LRSETPOSROUNDSFILT : LREAL;
	LRSETPOSROUNDSLAST : LREAL;
	LRTARGETPOSROUNDS : LREAL;
	XTARGETPOSVALID : BOOL;
	XTARGETPOSFROMMOVEREL : BOOL;
	LISETPOSCYCLE : LINT;
	LISETPOSCYCLERES : UDINT;
	XSETPOSCYCLEZERO : BOOL;
	XRECOVERLASTSETPOS_RAMP : BOOL := FALSE;
	XRECOVERLASTSETPOS_POSCTRL : BOOL := TRUE;
	XRECOVERYPOSVALID : BOOL;
	XMOVELASTSETPOS : BOOL;
	LRRECOVERYWINDOWPOS : LREAL;
	LRRECOVERYWINDOWNEG : LREAL;
	LRRECOVERYPOSITION : LREAL;
	LRRECOVERYVEL : LREAL := 360;
	LRRECOVERYACC : LREAL := 3600;
	LRRECOVERYDEC : LREAL := 3600;
	LRRECOVERYJERK : LREAL := 0;
	XSLSACTIVE : BOOL;
	XSLSACTIVEOLD : BOOL;
	XSLIREQUESTACTIVE : BOOL;
	XSWLIMITSACTIVE : BOOL;
	LRSLIDISTANCE : LREAL := 360;
	LRSLSVELOCITY : LREAL;
	LRSLSVELOCITYOLD : LREAL;
	LRSLSDECELERATION : LREAL;
	LRSLSDECELERATION2 : LREAL;
	LRSLSDECELERATIONOLD : LREAL;
	LRSLSJERK : LREAL;
	XSLSCHANGES : BOOL;
	XSLSNEWACTIVEDECELERATION : BOOL;
	WSLSWARNING : WORD;
	XLIMITERENABLEPOSITIVE : BOOL := TRUE;
	XLIMITERENABLENEGATIVE : BOOL := TRUE;
	XLIMITERENABLED : BOOL;
	XLIMITATIONSLSACTIVE : BOOL;
	XLIMITATIONACTIVE : BOOL;
	LRSLSDECTIME : LREAL := 100;
	LRSLSDECTIMEOLD : LREAL := 100;
	WSAFESTOPCONTROLWORD : WORD;
	WSAFESTOPCONTROLWORDOLD : WORD;
	READPARAMETER : L_DCO_ReadDriveParameter;
	WRITEPARAMETER : L_DCO_WriteDriveParameter;
	DWACTUALSPEEDCONTROLLERLIMIT : DWORD;
	XLIMITSPEEDCONTROLLERSLS : BOOL;
	DWDISABLESAFETYINTERFACE : DWORD;
	DWREQUESTSAFETYINTERFACE : DWORD;
	XFOLLOWERSLS : BOOL;
	LRSLSTIMER : LREAL;
	LRSLSTIMERTEMP : LREAL;
	XSLSACTIVATED : BOOL := FALSE;
	XSETSTOPBYDIRECTIONACTIVE : BOOL;
	XSETSTOPBYLIMITERACTIVE : BOOL;
	XSETSTOPCINHBYLIMITERACTIVE : BOOL;
	XSLSVELOCITYACTIVE : BOOL;
	XSLSDECTIMEACTIVE : BOOL;
	XSLSWARNINGACTIVE : BOOL;
	ETYPEFUNCTIONACT : L_MC1P_TypeFunction := L_MC1P_TypeFunction.Type_Any;
	SCSTOPBYERROR : L_MC1P_StopOperation;
	SCSTOPBYAXESGROUP : L_MC1P_StopOperation;
	DWAXISERRORITFID : DWORD := 0;
	ICMODE : WORD;
	ICMODEOLD : WORD;
	DWIC : DWORD;
	DWICOLD : DWORD;
	XINTERNALCONTROLMODEACTIVE : BOOL;
	XINTERNALCONTROLMODEACTIVEOLD : BOOL;
	XREFDUMMY : BOOL;
	LRREFDUMMY : LREAL;
	RREFDUMMY : REAL;
	WREFDUMMY : WORD;
	IREFDUMMY : INT;
	DWREFDUMMY : DWORD;
	DIREFDUMMY : DINT;
	LWREFDUMMY : LWORD;
	LIREFDUMMY : LINT;
	SREFDUMMY : STRING;
	USIREFDUMMY : USINT;
	BYREFDUMMY : BYTE;
	UIREFDUMMY : UINT;
	UDIREFDUMMY : UDINT;
	ULIREFDUMMY : ULINT;
	DWCALLCYCLE : DWORD;
	DWCALLCYCLE_US : DWORD;
	DWTPDELAYACTPOS : DWORD := 0;
	DWACTDCTIME : DWORD;
	PDWABSOLUTECOUNTER : POINTER TO DWORD;
	XGLOBALTIMESTAMPSUPPORTED : BOOL;
	HMOTIONTASK : SysTypes.RTS_IEC_HANDLE := 0;
	WACTPOSIDX : WORD;
	ADWACTTIMESTAMPS : ARRAY [0..15] OF DWORD;
	ALRACTPOSITION : ARRAY [0..15] OF LREAL;
	ALRACTPOSITIONUNFILTERED : ARRAY [0..15] OF LREAL;
	ALRACTPOSROUNDS : ARRAY [0..15] OF LREAL;
	ALRTPPOSOFFSET : ARRAY [0..15] OF LREAL;
	HEVENTRESETOCCURED : SysTypes.RTS_IEC_HANDLE := SysTypes.RTS_INVALID_HANDLE;
	HINTERFACERESETOCCURED : SysTypes.RTS_IEC_HANDLE := SysTypes.RTS_INVALID_HANDLE;
	XGENERRORREAKTINDEVICE : BOOL;
	XFORWARDERRORSASWARNINGS : BOOL;
	WEVTCOUNT_SETERRORREACTION : WORD;
	WEVTCOUNT_UPDATEACTIVEERROR : WORD;
	WEVTCOUNT_RESETOCCURED : WORD;
	XINTERNALERRORRESET : BOOL;
	XINTERNALERRORRESETFROMLEM : BOOL;
	WHANDLINGLEM : WORD := 0;
	XERRORRESETREQUESTSEND : BOOL;
	WERRORRESETREQUESTSEND : WORD := 0;
	RESETINTERNAL : L_MC1P_Reset_Internal;
	DWACTSTATEDETERMINEEVENT : DWORD;
	SEVERITYCMDEXT : USINT;
	EERRORREACTIONCMDEXT : L_IE1P_SeverityLevel := L_IE1P_SeverityLevel.NO_RESPONSE;
	DWERRORINFOEXT : DWORD;
	XEXTERROR : BOOL;
	MYSYSTEMSEVERITY : USINT;
	XJOGGINGACTIVE : BOOL;
	LRJOGGINGSETVEL : LREAL := 360.0;
	LRJOGGINGSETACC : LREAL := 360.0;
	LRJOGGINGSETDEC : LREAL := 1440.0;
	LRJOGGINGSETJERK : LREAL := 0.0;
	XJOGUSEAXISPAR : BOOL := FALSE;
	XHOMEPOSUSEAXISPAR : BOOL := FALSE;
	XUSEFASTSTOPBEHAVIOUR : BOOL := TRUE;
	XFIRSTBASEINITDONE : BOOL := FALSE;
	EHWLIMITERRORREACTION : USINT := 19;
	ESWLIMITERRORREACTION : USINT := 19;
	ELIMITPROFILEERRORREACTION : USINT := 2;
	ECINHERRORREACTION : USINT := 19;
	LRREFROUNDS : LREAL;
	XMOVELASTSETPOSACTIVE : BOOL;
	XSTAYINLASTSTATEACTIVE : BOOL;
	XABORTSTAYINLASTSTATEREQUEST : BOOL;
	XCINHACTIVE : BOOL;
	XCINHACTIVEOLD : BOOL;
	XSTOACTIVEOLD : BOOL;
	XSETPOSINSIDEWINDOW : BOOL;
	XSTAYINLASTSTATEACTIVEOLD : BOOL;
	XDRIVESTATEBEFORECINH : BOOL;
	LRPOSOFFSETMOVELASTSETPOS : LREAL;
	LRVELOFFSETMOVELASTSETPOS : LREAL;
	LRACCOFFSETMOVELASTSETPOS : LREAL;
	XHALTPARAMETERSUPPORTED : BOOL;
	LRHALTDEC : LREAL := 1800;
	LRHALTJERK : LREAL := 0;
	XHALTBYABC : BOOL;
	SCTIMESTAMP : L_MC1P_TimeStamp;
	XACTIVATETIMEMEASUREMENT : BOOL;
	XISSAFETYDEVICE : BOOL;
	WINDEXINT : WORD;
	BYSUBINDEXINT : BYTE;
	BYSLSREADWRITECOUNTER : BYTE;
	XCALCMODULOASLIMITED : BOOL := FALSE;
	FBSTEADYSTATE : L_MC1P_SteadyState;
	WDEVICETYPETEMP : WORD;
	DWIODRVDEVICEIDTEMP : DWORD;
	XUSEQSPDRIVEINSTEADOFQSPAPPL : BOOL := FALSE;
	XMINJERKAVAILABLE : BOOL;
	XMINJERKAVAILABLEOLD : BOOL;
	XMINJERKACTIVE : BOOL;
	XMINJERKACTIVEOLD : BOOL;
	LRMINJERK : LREAL;
	LRMINJERKOLD : LREAL;
	LRMOVEVELOFFSETVELOLD : LREAL;
	XSETVALUESFORINTERNALSTOPAVAILABLE : BOOL;
	XSETVALUESFROMINTERNALSTOPACTIVE : BOOL;
	XOPTRAMPSFORMANUALJOG : BOOL := TRUE;
	XCHANGECINHPARNOTALLOWED : BOOL := FALSE;
	XBEHAVIOURFORVIRTUALMASTER : BOOL := FALSE;
	STOPAXISBYERRORREACTIONCOUNTER : L_IE1P_ReactionCounter;
	SCSTOPAXISBYERRORREACTION : L_MC1P_StopOperation;
	MODULEHANDLERBASE : L_IMHP_ModuleHandler := STRUCT(CompActiveDefault := FALSE, Layer := L_IMHP_Layer.Motion, CompType := L_IMHP_ComponentType.VirtualAxis);
	FB_GETDIRECTIONACTVALUES : L_MC1P_GetDirection;
	WDIRECTIONSETVALUES : WORD;
	XQSPWITHOUTREACTION : BOOL;
	XVALIDMFEFWVERSION : BOOL;
	XSETDRIVEQSPDISABLED : BOOL;
	EKINDOFMOTIONSELECTION : L_MC1P_KindOfMotion;
	EACTIVEUNIT : WORD;
	WERRORIDINITSTATE : WORD;
	ITFMANIPULATEACTVALUES : L_Mc1P_IManipulateActValues;
	XSETVELOCITYGTSLS : BOOL;
	XCLOSEBRAKEATQSPRAMPEND : BOOL;
	C_STRNOERROR : STRING := '-';
	C_STRUNDEFERROR : STRING := 'undefined';
	C_MAXFILTER : WORD := 2;
	C_MAXCOMP : WORD := 2;
	C_MAXFILTERINT : WORD := (c_MaxFilter + 1);
	C_UDILOGCOMPONENDID : UDINT := 16#2800;
	ACTACCELERATION : LREAL;
	ACTPOSITION : LREAL;
	ACTTORQUE : LREAL;
	ACTVELOCITY : LREAL;
	AXISPOOLCOUNT : WORD;
	AXISSLOT : L_MC1P_AxisSlot;
	CIA402ADVANCEDAXIS : BOOL;
	CMDCINH : BOOL;
	CMDFASTSTOP : BOOL;
	CMDFASTSTOPCINH : BOOL;
	CMDQSP : BOOL;
	CMDQSPCINH : BOOL;
	CYCLELENGTH : LREAL;
	FEEDCONSTANT : LREAL;
	GETACTIVELIMTERCONTROLWORD : DWORD;
	GETMASTERID : POINTER TO BYTE;
	HOMEPOSPERMANTENTSETACTIVE : BOOL;
	HOMEPOSPERMANTENTSETACTIVELOADENCODER : BOOL;
	LICENSECONFIG : STRING;
	MODULEHANDLER : L_IMHP_IModuleHandler;
	QSPATFASTSTOPEND : BOOL;
	QSPWITHOUTREACTION : BOOL;
	RESETFOLLOWINGERRORATFASTSTOPEND : BOOL;
	SERVICEDIRECTION : L_MC1P_ServiceDirection;
	SETACCELERATIONFORSYNC : LREAL;
	SETHOMEPOSSTATEINDEPENDENTACTIVE : BOOL;
	SETPOSITIONFORSYNC : LREAL;
	SETPOSROUNDS : LREAL;
	SETTORQUEFORSYNC : LREAL;
	SETVELOCITYFORSYNC : LREAL;
	STARTPOSFORINTERNALSTOP : LREAL;
	TASKCYCLE : LREAL;
	TIMEDELAYACTPOS : LREAL;
	TIMEDELAYSETPOS : LREAL;
	TRAVERSINGRANGE : L_MC1P_TraversingRange;
	USEDASINTERNALAXISINSTANCE : BOOL;
	USEDBYVIRTUALMASTER : BOOL;
END_VAR
END_FUNCTION_BLOCK

METHOD ACTIVATEACYCLICMODE
VAR_INPUT
	XACTIVATE : BOOL;
END_VAR
END_METHOD

METHOD CALCACTDIRECTION
END_METHOD

METHOD CALCACTPOSUNFILTERED : LREAL
END_METHOD

METHOD CALCSETDIRECTION : WORD
VAR_INPUT
	LRCYCVELIN : LREAL;
END_VAR
END_METHOD

METHOD CALLSIMULATION
VAR_INPUT
	CALLSTATE : L_UBUP_StateHandleCase;
END_VAR
END_METHOD

METHOD CHECKDIRECTION : BOOL
VAR_INPUT
	DIRECTION : MC_DIRECTION;
	ETYPEFUNCTION : L_MC1P_TypeFunction;
END_VAR
END_METHOD

METHOD CHECKMAXMODULOPOSDIFF
END_METHOD

METHOD CHECKPLNOTVALID : BOOL
END_METHOD

METHOD CHECKPLAUSIBILITYOFSETVALUES
END_METHOD

METHOD CHECKPOWER : BOOL
VAR_INPUT
	DWPOSSTATE : DWORD;
	LRVEL : LREAL;
END_VAR
END_METHOD

METHOD CHECKSLSVELOCITY : BOOL
END_METHOD

METHOD CHECKSETPOSINWINDOW : BOOL
END_METHOD

METHOD COMPENSATELOADPOSOFFSET
END_METHOD

METHOD ENABLEDRIVE : BOOL
VAR_INPUT
	XENABLE : BOOL;
END_VAR
END_METHOD

METHOD FLOATTOFRAC
VAR_INPUT
	LRINPUT : LREAL;
	PDIINTEGER : POINTER TO DINT;
	PUDIRESIDUAL : POINTER TO UDINT;
END_VAR
END_METHOD

METHOD FLOATTOFRACLINT
VAR_INPUT
	LRINPUT : LREAL;
	PLIINTEGER : POINTER TO LINT;
	PUDIRESIDUAL : POINTER TO UDINT;
END_VAR
END_METHOD

METHOD GENACTVALUES
END_METHOD

METHOD GETACTVEL : LREAL
END_METHOD

METHOD GETACTVELOCITYEXACT : LREAL
END_METHOD

METHOD GETACTIVEQUICKSTOPOPTION : L_MC1P_QuickStopOption
END_METHOD

METHOD GETAXISSLOT : UINT
END_METHOD

METHOD GETBRAKE : POINTER TO L_MC1P_BrakeControlBase
END_METHOD

METHOD GETBRAKESERVICE : POINTER TO L_MC1P_BrakeService
END_METHOD

METHOD GETCOUPLEDMASTERAXIS : POINTER TO BYTE
END_METHOD

METHOD GETCOUPLEDPHASINGMASTERAXIS : POINTER TO BYTE
END_METHOD

METHOD GETDRIVESTATE : BOOL
END_METHOD

METHOD GETEFFECTIVEMFESPEEDOFFSET : INT
VAR_INPUT
	INOFFSET : INT;
END_VAR
END_METHOD

METHOD GETMODULODIFF : LREAL
VAR_INPUT
	LRDIFF : LREAL;
END_VAR
VAR_IN_OUT
	AXIS : AXIS_REF;
END_VAR
END_METHOD

METHOD GETMODULOPOSITION : LREAL
VAR_INPUT
	LRNEWPOS : LREAL;
END_VAR
VAR_OUTPUT
	LRROUNDS : LREAL;
END_VAR
VAR_IN_OUT
	AXIS : AXIS_REF;
END_VAR
END_METHOD

METHOD GETPGMOVE : REFERENCE TO L_MC1P_PosProfiler
VAR_INPUT
	ITFPGACTIVE : L_MC1P_IPosProfilerActive;
END_VAR
END_METHOD

METHOD GETPGDUMMY : REFERENCE TO L_MC1P_PosProfiler
END_METHOD

METHOD GETPGSUPER : REFERENCE TO L_MC1P_PosProfiler
VAR_INPUT
	ITFPGACTIVE : L_MC1P_IPosProfilerActive;
END_VAR
END_METHOD

METHOD GETPHASESHIFT
VAR_OUTPUT
	LRPOS : LREAL;
	LRVEL : LREAL;
	LRACC : LREAL;
END_VAR
END_METHOD

METHOD GETRECEIVEDATA : DWORD
VAR_INPUT
	LWMASK : LWORD;
END_VAR
END_METHOD

METHOD GETTPWITHPOSITIONACTIVE : BOOL
VAR_INPUT
	SITPNUMBER : SINT;
END_VAR
END_METHOD

METHOD GETTPWITHTIMESTAMPACTIVE : BOOL
VAR_INPUT
	SITPNUMBER : SINT;
END_VAR
END_METHOD

METHOD HALTCALLEDBYABC
VAR_INPUT
	XCALLEDBYABC : BOOL;
END_VAR
END_METHOD

METHOD HLP_MODULOPOS : LREAL
VAR_INPUT
	LRPOSITION : LREAL;
	LRCYCLELENGTH : LREAL;
END_VAR
END_METHOD

METHOD HLP_MODULOPOS2 : LREAL
VAR_INPUT
	LRPOSITION : LREAL;
	LRCYCLELENGTH : LREAL;
	LRINVCYCLELENGTH : LREAL;
END_VAR
END_METHOD

METHOD INTOLERANCEWINDOW : BOOL
VAR_INPUT
	LRPOSITION : LREAL;
END_VAR
VAR_OUTPUT
	DIRECTION : MC_DIRECTION;
END_VAR
END_METHOD

METHOD INTERNALCONTROLMODE
END_METHOD

METHOD ISINCLUDEDINRECEIVEDATA : BOOL
VAR_INPUT
	LWMASK : LWORD;
END_VAR
END_METHOD

METHOD ISINCLUDEDINTRANSMITDATA : BOOL
VAR_INPUT
	LWMASK : LWORD;
END_VAR
END_METHOD

METHOD ISMOTIONALLOWED : BOOL
VAR_INPUT
	ETYPEFUNCTION : L_MC1P_TypeFunction;
END_VAR
VAR_IN_OUT
	XSUPERIMPOSED : BOOL;
END_VAR
END_METHOD

METHOD ISMOTIONALLOWED2 : BOOL
VAR_INPUT
	ETYPEFUNCTION : L_MC1P_TypeFunction;
	XCHECKHOMEPOS : BOOL;
END_VAR
VAR_OUTPUT
	EERRORCAUSE : L_IE1P_Error := L_IE1P_Error.NoError;
END_VAR
VAR_IN_OUT
	XSUPERIMPOSED : BOOL;
END_VAR
END_METHOD

METHOD LEAVESERVICESTATE
END_METHOD

METHOD LEAVESERVICESTATEBEAVIOUR : DINT
VAR_INPUT
	XDISABLEDRIVE : BOOL;
END_VAR
END_METHOD

METHOD LEAVESERVICESTATESTART : BOOL
END_METHOD

METHOD LIMITPROFILEDATA : WORD
VAR_INPUT
	PPROFLE : POINTER TO L_MC1P_ProfileParameter;
	PPROFLEOLD : POINTER TO L_MC1P_ProfileParameter;
END_VAR
END_METHOD

METHOD LOCKEDFORSINGLEMOTION
VAR_INPUT
	XLOCKED : BOOL;
END_VAR
END_METHOD

METHOD REGISTERAXESGROUP : BOOL
VAR_INPUT
	XUNREGISTER : BOOL;
	PAXESGROUP : POINTER TO BYTE;
END_VAR
END_METHOD

METHOD REGISTERFUNCTION : WORD
END_METHOD

METHOD REGISTERPHASINGFUNCTION : WORD
VAR_INPUT
	PMASTERAXIS : POINTER TO BYTE;
END_VAR
END_METHOD

METHOD REGISTERSUPERFUNCTION : WORD
END_METHOD

METHOD REGISTERSYNCFUNCTION : WORD
VAR_INPUT
	PMASTERAXIS : POINTER TO BYTE;
END_VAR
END_METHOD

METHOD RESETERRORSTATEOFCOMMANDS : BOOL
END_METHOD

METHOD RESETFOLLOWINGERROR
END_METHOD

METHOD RESETMOVEBUFFEREDINFO
END_METHOD

METHOD RESETMOVEINFO
END_METHOD

METHOD SERVICEMODEHANDLINGINDRIVEACTIVE : BOOL
END_METHOD

METHOD SETACTPOSITION
VAR_INPUT
	POSITION : LREAL;
	RELATIVE : BOOL;
END_VAR
END_METHOD

METHOD SETAXISSTATUSWORD
END_METHOD

METHOD SETBUFFERDATAALLOWED : BOOL
VAR_INPUT
	EMODE : MC_BUFFER_MODE;
	LRSPEED1 : LREAL;
	LRSPEED2 : LREAL;
	DWINSTANCE : __XWORD;
END_VAR
END_METHOD

METHOD SETDCBRAKE
VAR_INPUT
	XSETDCBRAKE : BOOL;
END_VAR
VAR_OUTPUT
	XDCBRAKEACTIVE : BOOL;
END_VAR
END_METHOD

METHOD SETENCODERITF
VAR_INPUT
	ENCODERIN : L_MC1P_IEncoderInterface;
END_VAR
END_METHOD

METHOD SETHOMEABSSWITCH
VAR_INPUT
	HOMEABSSWITCH : BOOL;
END_VAR
END_METHOD

METHOD SETHOMEABSSWITCHOVERWRITE
VAR_INPUT
	XHOMEABSSWITCHSIGNAL : BOOL;
	XOVERWRITESIGNAL : BOOL;
END_VAR
END_METHOD

METHOD SETMACHINEDATA
END_METHOD

METHOD SETPHASESHIFT
VAR_INPUT
	LRPOS : LREAL;
	LRVEL : LREAL;
	LRACC : LREAL;
END_VAR
END_METHOD

METHOD SETPOSEQACTPOS
END_METHOD

METHOD SETPRECONTROLMODE
VAR_INPUT
	EPRECONTROLMODENEW : L_MC1P_PreControlMode := L_MC1P_PreControlMode.Automatic;
END_VAR
END_METHOD

METHOD SETTARGETPOS
VAR_INPUT
	LRTARGETPOSNEW : LREAL;
	LRTARGETPOSROUNDSNEW : LREAL;
	XVALID : BOOL;
END_VAR
END_METHOD

METHOD SETTARGETPOS2
VAR_INPUT
	LRTARGETPOSNEW : LREAL;
	LRTARGETPOSROUNDSNEW : LREAL;
	XVALID : BOOL;
	XRELMODE : BOOL;
END_VAR
END_METHOD

METHOD SETTORQUEVALUE
VAR_INPUT
	LRTORQUE : LREAL;
	WMODE : WORD;
END_VAR
END_METHOD

METHOD SETVELEQREFVALUE
VAR_INPUT
	LRREFVELOCITY : LREAL;
END_VAR
END_METHOD

METHOD SETVELOCITYOFFSET
VAR_INPUT
	WMODE : WORD;
	LROFFSETVELOCITY : LREAL;
END_VAR
END_METHOD

METHOD SPEEDEQZERO : BOOL
VAR_INPUT
	LRSPEEDIN : LREAL;
END_VAR
END_METHOD

METHOD SUSPENDFOLLOWINGERROR
VAR_INPUT
	XSUSPEND : BOOL;
END_VAR
END_METHOD

METHOD UPDATEERRORINFO
END_METHOD

METHOD UPDATEREADYFORMOTIONSTATUS : BOOL
VAR_INPUT
	AXISENABLED : BOOL;
END_VAR
END_METHOD

METHOD CALLRECIEVEPARAMETER
END_METHOD

METHOD CALLSDODATAHANDLING
END_METHOD

METHOD CALLTRANSMITPARAMETER
END_METHOD

METHOD CHECKCOMMUNCATION
END_METHOD

METHOD CHECKMAPPEDDATAVALID : BOOL
VAR_INPUT
	PADDDATA : POINTER TO BYTE;
	PDATA : POINTER TO POINTER TO BYTE;
END_VAR
VAR_OUTPUT
	XERROR : BOOL;
	EERRORID : L_IE1P_Error;
END_VAR
END_METHOD

METHOD GETMAPPEDDATA : POINTER TO BYTE
VAR_INPUT
	UIINDEX : WORD;
	USISUBINDEX : USINT;
	USISIZE : USINT;
	XWRITEACCESS : BOOL;
	PADDDATA : POINTER TO BYTE;
	PXWAITFORINITACCESS : POINTER TO BOOL;
END_VAR
VAR_OUTPUT
	EERRORID : L_IE1P_Error;
	XERROR : BOOL;
	USISIZEACT : USINT := 0;
END_VAR
END_METHOD

METHOD GETMAPPEDDATASUPPORT : BOOL
END_METHOD

METHOD RESETMAPPEDDATA
VAR_INPUT
	PADDDATA : POINTER TO BYTE;
END_VAR
END_METHOD

METHOD RESETSDODATA : DINT
VAR_INPUT
	IDX : DWORD;
	PDWSEMAPARACCESS : POINTER TO DWORD;
END_VAR
VAR_IN_OUT
	SDODATA : L_DCO_SdoData;
END_VAR
END_METHOD

METHOD CONFIGUREAXIS
END_METHOD

METHOD CONFIGUREAXIS2
END_METHOD

METHOD CONFIGUREAXISCONNECTOR
END_METHOD

METHOD CONFIGUREAXISCONNECTORBASICS : BOOL
END_METHOD

METHOD CONNECTCMDITFAUTOTUNING
END_METHOD

METHOD DETERMINETASKCYCLEINTERVAL : UDINT
END_METHOD

METHOD ENABLEAXISCONNECTOR : BOOL
END_METHOD

METHOD FINDANDCONNECTMOTIONUTILS
END_METHOD

METHOD GETTRANSMITCYCLESACTPOSFORPOSCTRL : LREAL
END_METHOD

METHOD REGISTERAXISPROPERTIES
END_METHOD

METHOD RESETAXISCONNECTOR
END_METHOD

METHOD SETAXISPROPERTIES
VAR_INPUT
	XUSEVIRTUAL : BOOL;
END_VAR
END_METHOD

METHOD UPDATEFATHERCONNECTOR
END_METHOD

METHOD CHECKAVAILABLECONTROLMODE : BOOL
END_METHOD

METHOD CONFIGURECONTROLMODE
VAR_OUTPUT
	EERRORID : L_IE1P_Error;
END_VAR
END_METHOD

METHOD GETDEFAULTCONTROLMODE : L_MC1P_ControlMode
END_METHOD

METHOD ISAVAILABLECONTROLMODE : BOOL
VAR_INPUT
	ECONTROLMODE : L_MC1P_ControlMode;
END_VAR
VAR_OUTPUT
	EERRORID : L_IE1P_Error;
END_VAR
END_METHOD

METHOD SETCONTROLMODE : BOOL
VAR_INPUT
	ECONTROLMODE : L_MC1P_ControlMode := L_MC1P_ControlMode.PosCtrlDrive;
	XKEEPACTPOSPRIORFDB : BOOL := FALSE;
	XRESTARTPOSITIONING : BOOL := FALSE;
END_VAR
VAR_OUTPUT
	EERRORID : L_IE1P_Error;
END_VAR
END_METHOD

METHOD SETCONTROLERITF
VAR_INPUT
	ITFCONTROLERNEW : L_MC1P_IControllerInterface;
END_VAR
END_METHOD

METHOD SETDEFAULTCONTROLMODE : BOOL
END_METHOD

METHOD CLEARERROR
VAR_INPUT
	PINSTANCE : POINTER TO BYTE := 0;
END_VAR
END_METHOD

METHOD CLEARERROR2
VAR_INPUT
	INSTANCEID : DWORD := 0;
END_VAR
END_METHOD

METHOD CLEARERRORID
VAR_INPUT
	PINSTANCE : POINTER TO BYTE := 0;
	WERRORID : WORD;
END_VAR
END_METHOD

METHOD CLEARERRORID2
VAR_INPUT
	INSTANCEID : DWORD := 0;
	WERRORID : WORD;
END_VAR
END_METHOD

METHOD CLEARERRORID3
VAR_INPUT
	INSTANCEID : DWORD := 0;
	WERRORID : WORD;
	DWEXTENDEDERRORINFO : DWORD;
END_VAR
END_METHOD

METHOD GETERRORITFID : DWORD
END_METHOD

METHOD HANDLEERRORENTRY : BOOL
VAR_INPUT
	WERRORID : L_IE1P_Error := 0;
	INSTANCEID : DWORD := 0;
	PSINSTANCENAME : POINTER TO BYTE := 0;
	DWEXTENDEDERRORINFO : DWORD;
	EERRORREACTION : L_IE1P_SeverityLevel := 0;
	XAUTORESET : BOOL;
	XNOLOGGINGENTRY : BOOL;
	XEXTERNALERROR : BOOL;
END_VAR
END_METHOD

METHOD NOTIFYERROR : BOOL
VAR_INPUT
	WERRORID : L_IE1P_Error := 0;
	PINSTANCE : POINTER TO BYTE := 0;
	PSINSTANCENAME : POINTER TO BYTE := 0;
	XSETERRORSTOP : BOOL := FALSE;
END_VAR
END_METHOD

METHOD NOTIFYERROR2 : BOOL
VAR_INPUT
	WERRORID : L_IE1P_Error := 0;
	INSTANCEID : DWORD := 0;
	PSINSTANCENAME : POINTER TO BYTE := 0;
	EERRORREACTION : L_IE1P_SeverityLevel := 0;
END_VAR
END_METHOD

METHOD SERERRORREACTIONEXTERN
VAR_INPUT
	EERRORREACTION : L_IE1P_SeverityLevel;
	WERRORID : WORD;
	INSTANCEID : DWORD := 0;
	XAUTORESET : BOOL;
	DWEXTENDEDERRORINFO : DWORD;
	XEXTERNALERROR : BOOL;
END_VAR
END_METHOD

METHOD UPDATEERRORREAKTION
VAR_INPUT
	SEVERITY : L_IE1P_SeverityLevel;
END_VAR
END_METHOD

METHOD EVENTCALLBACK : UDINT
VAR_INPUT
	PEVENTPARAM : POINTER TO EventParam;
END_VAR
END_METHOD

METHOD REGISTEREVENT
END_METHOD

METHOD UNREGISTEREVENT
END_METHOD

METHOD RESETHOMEPOS
END_METHOD

METHOD RESETHOMEPOS2
VAR_INPUT
	ERESETINFO : L_IE1P_Error;
END_VAR
END_METHOD

METHOD RESETHOMEPOSLOADENCODER
VAR_INPUT
	ERESETINFO : L_IE1P_Error;
END_VAR
END_METHOD

METHOD SETHOMEPOSDEPENDONMODESTATEINDEPENDENT : BOOL
VAR_INPUT
	EHOMEMODE : L_MC1P_HomeMode;
	LRPOSITION : LREAL;
	LROFFSETPOSITION : LREAL;
	EHOMEPOSINFO : L_IE1P_Error;
END_VAR
VAR_OUTPUT
	XERROR : BOOL;
	EERRORID : L_IE1P_Error;
END_VAR
END_METHOD

METHOD SETHOMEPOSITION
VAR_INPUT
	POSITION : LREAL;
	RELATIVE : BOOL;
	XRESTARTPOSITIONING : BOOL := FALSE;
END_VAR
END_METHOD

METHOD SETHOMEPOSITION2
VAR_INPUT
	POSITION : LREAL;
	RELATIVE : BOOL;
	XRESTARTPOSITIONING : BOOL := FALSE;
	EHOMEPOSINFO : L_IE1P_Error;
END_VAR
END_METHOD

METHOD SETHOMEPOSITIONWITHMODROUNDS
VAR_INPUT
	POSITION : LREAL;
	RELATIVE : BOOL;
	ROUNDS : LREAL;
	XRESTARTPOSITIONING : BOOL;
	EHOMEPOSINFO : L_IE1P_Error;
END_VAR
END_METHOD

METHOD ITFCHECKERRORRESETOCCURED : BOOL
VAR_IN_OUT
	RESETTIME : SYSTIME;
END_VAR
END_METHOD

METHOD ITFCLEARERROR : DWORD
VAR_INPUT
	ESEVERITY : L_IE1P_SeverityLevel;
	WERRORID : WORD;
	WCOMPID : WORD;
	DWINSTANCEID : DWORD := 0;
END_VAR
END_METHOD

METHOD ITFCLEARREACTION
VAR_INPUT
	EREACTION : L_IE1P_Reaction;
	DICLEARCOUNT : DINT;
	DWINSTANCEID : DWORD;
END_VAR
END_METHOD

METHOD ITFGETACTUALERRORCODE : DWORD
VAR_OUTPUT
	ESEVERITY : WORD;
END_VAR
END_METHOD

METHOD ITFREGISTERERRORINSTANCE : DWORD
END_METHOD

METHOD ITFRESETACTIVE : BOOL
END_METHOD

METHOD ITFRESETERROR : DWORD
VAR_INPUT
	ERRORHANDLE : SysTypes.RTS_IEC_HANDLE := 0;
END_VAR
END_METHOD

METHOD ITFRESETERRORREACTION
VAR_INPUT
	DWINSTANCEID : DWORD := 0;
END_VAR
END_METHOD

METHOD ITFSETERROR : DWORD
VAR_INPUT
	ESEVERITY : L_IE1P_SeverityLevel;
	WERRORID : WORD;
	WCOMPID : WORD;
	DWINSTANCEID : DWORD := 0;
	EREACTION : L_IE1P_Reaction;
END_VAR
END_METHOD

METHOD GETDIRECTION : WORD
VAR_INPUT
	VALUESOURCE : MC_SOURCE;
END_VAR
END_METHOD

METHOD GETMASTERERROR : BOOL
VAR_OUTPUT
	EERRORID : L_IE1P_Error;
END_VAR
END_METHOD

METHOD GETSTEADYSTATE : POINTER TO L_MC1P_SteadyState
END_METHOD

METHOD GETAXISFROMPOOL : POINTER TO AXIS_REF
VAR_INPUT
	WINDEX : WORD;
END_VAR
END_METHOD

METHOD CHECKINPOSITION
END_METHOD

METHOD SETINPOSITION
VAR_INPUT
	XDONE : BOOL;
	LRINTARGETPOSITION : LREAL;
END_VAR
END_METHOD

METHOD ACTIVATESS1
END_METHOD

METHOD CALCULATE_DECELERATION : LREAL
VAR_INPUT
	LRJERK : LREAL;
	LRTOTALTIME : LREAL;
	LRACTVEL : LREAL;
	LRTARGETVEL : LREAL;
	LRACCMAX : LREAL;
END_VAR
END_METHOD

METHOD CHECKLIMITERREQUESTS
END_METHOD

METHOD CHECKSLSCHANGES : BOOL
VAR_OUTPUT
	XLIMITERCONTROLCHANGED : BOOL;
	XSLSPARAMETERCHANGED : BOOL;
	XSLSNEWACTIVEDECELERATION : BOOL;
END_VAR
END_METHOD

METHOD CHECKSAFETYOPTIONAVAILABLE : BOOL
VAR_INPUT
	DWPRODUCTCODE : DWORD;
END_VAR
END_METHOD

METHOD LIMITSPEEDCONTROLLER
END_METHOD

METHOD PROCESSSSX
VAR_INPUT
	DWCONTROL : DWORD;
END_VAR
END_METHOD

METHOD UPDATEACTIVESLSSETVEL
VAR_INPUT
	LRVEL : LREAL;
END_VAR
END_METHOD

METHOD CHECKHWLIMITS : BOOL
END_METHOD

METHOD CHECKLIMITCHANGES : BOOL
VAR_OUTPUT
	XPOSSWLIMITCHANGED : BOOL;
	XNEGSWLIMITCHANGED : BOOL;
END_VAR
END_METHOD

METHOD CHECKMAXVALUES : BOOL
VAR_INPUT
	VELOCITY : LREAL;
	ACCELERATION : LREAL;
	JERK : LREAL;
END_VAR
END_METHOD

METHOD CHECKSWLIMITS : BOOL
VAR_INPUT
	XSETERRORSTOP : BOOL;
END_VAR
END_METHOD

METHOD DISABLESWLIMIT
VAR_INPUT
	XDISABLE : BOOL;
END_VAR
END_METHOD

METHOD GETACTDIRECTION : MC_DIRECTION
VAR_INPUT
	XCALCULATE : BOOL;
END_VAR
END_METHOD

METHOD GETSWLIMITSACTIVE : BOOL
END_METHOD

METHOD CALCCYCLELENGTH
END_METHOD

METHOD CALCULATESCALING : BOOL
END_METHOD

METHOD GETVIRTUAL : BOOL
END_METHOD

METHOD MACHINEDATACHANGED : BOOL
END_METHOD

METHOD WRITENEWMACHINEDATA
VAR_INPUT
	LRFEEDCONSTANTNEW : LREAL := 360.0;
	DWGEARDENOMINATORNEW : DWORD := 1;
	DWGEARNUMERATORNEW : DWORD := 1;
	DWADDGEARDENOMINATORNEW : DWORD := 1;
	DWADDGEARNUMERATORNEW : DWORD := 1;
	DWPOSRESOLUTIONNEW : DWORD := 65536;
	XORIENTATIONNEW : BOOL := FALSE;
	ETRAVERSINGRANGENEW : L_MC1P_TraversingRange := L_MC1P_TraversingRange.Limited;
	LRCYCLELENGTHNEW : LREAL := 360.0;
END_VAR
END_METHOD

METHOD COMPAREAXISNAME : BOOL
VAR_IN_OUT
	SAXISNAME : STRING;
END_VAR
END_METHOD

METHOD GETAXIS : POINTER TO AXIS_REF
END_METHOD

METHOD CALCSCALEFUNCTIONS
VAR_INPUT
	OFFSET : DWORD;
	INDEX : WORD;
END_VAR
END_METHOD

METHOD SETMACHINEDATAPARAMETER
END_METHOD

METHOD CALLCOMPFUNCTIONS
VAR_OUTPUT
	XCOMPERROR : BOOL;
END_VAR
END_METHOD

METHOD CALLFILTERFUNCTIONS
VAR_OUTPUT
	XFILTERERROR : BOOL;
END_VAR
END_METHOD

METHOD CHECKSETVALUESAVAILABLE
END_METHOD

METHOD RESETSETVALUESAVAILABLE
END_METHOD

METHOD RESTORESETVALUES
END_METHOD

METHOD SETCOMPITF : WORD
VAR_INPUT
	EINDEX : WORD;
	ITFCOMP : L_MC1P_ICompensationInterface;
END_VAR
END_METHOD

METHOD SETFILTERITF : WORD
VAR_INPUT
	EINDEX : WORD;
	ITFFILTER : L_MC1P_ISetvalueManipulationInterface;
	XFILTERINTERNALSET : BOOL;
END_VAR
END_METHOD

METHOD SETSETVALUESAVAILABLE
END_METHOD

METHOD SUSPENDSETVALUEFILTERCALL
VAR_INPUT
	XSUSPENDSETVALUEFILTERCALL : BOOL;
END_VAR
END_METHOD

METHOD ABORTACTIVEFUNCTION
END_METHOD

METHOD DRIVEQSP
END_METHOD

METHOD ERRORSTOP
END_METHOD

METHOD INTERNALSTOP : BOOL
VAR_INPUT
	XSTOP : BOOL;
	ESETSTATE : L_MC1P_AXIS_STATE;
	XPOSMODE : BOOL := FALSE;
	LRTARGETPOS : LREAL := 0;
	XABORTACTIVEFUNCTION : BOOL := TRUE;
END_VAR
VAR_IN_OUT
	XSTOPACTIVE : BOOL;
	XSTOPDONE : BOOL;
END_VAR
END_METHOD

METHOD MOVEBACKTOLASTSETPOS : BOOL
VAR_INPUT
	XSTOP : BOOL;
END_VAR
VAR_IN_OUT
	XSTOPACTIVE : BOOL;
	XSTOPDONE : BOOL;
END_VAR
END_METHOD

METHOD RAMPDOWN
END_METHOD

METHOD RAMPQSP
VAR_INPUT
	CALLEDFROMAPP : BOOL;
END_VAR
END_METHOD

METHOD RESETRAMPDOWN
END_METHOD

METHOD SETAXISSTOPINT : BOOL
VAR_INPUT
	XSTOP : BOOL;
	SCSTOPCMD : L_MC1P_StopOperation;
END_VAR
END_METHOD

METHOD SETFASTSTOPINT : BOOL
VAR_INPUT
	XSTOP : BOOL;
END_VAR
END_METHOD

METHOD SETSTANDSTILLSTATE
VAR_INPUT
	XRAMPDOWN : BOOL;
END_VAR
END_METHOD

METHOD STARTRAMPDOWN
END_METHOD

METHOD HLP_GETPARAMETER : BOOL
END_METHOD

METHOD HLP_GETPARAMETERPROPERTIES : BOOL
VAR_INPUT
	DIPARAMETER : DINT;
END_VAR
VAR_OUTPUT
	PPARAMADDR : POINTER TO BYTE := 0;
	EORDINALTYPE : L_MC1P_OrdinalType := L_MC1P_OrdinalType.otNONE;
	XREADWRITE : BOOL := FALSE;
	LRUNITFACTOR : LREAL := 1.0;
	LRDEFAULTVALUE : LREAL := 0.0;
	WVALUERANGES : WORD := 0;
	PVALUERANGES : POINTER TO L_MC1P_MinMaxValue := 0;
END_VAR
END_METHOD

METHOD HLP_INITPARREF
END_METHOD

METHOD HLP_READBOOLPARAMETER : BOOL
VAR_INPUT
	PARAMETER : DINT;
	PXVALUE : POINTER TO BOOL;
END_VAR
END_METHOD

METHOD HLP_READPARAMETER : BOOL
VAR_INPUT
	PARAMETER : DINT;
	PLRVALUE : POINTER TO LREAL;
END_VAR
END_METHOD

METHOD HLP_WRITEBOOLPARAMETER : BOOL
VAR_INPUT
	PARAMETER : DINT;
	PXVALUE : POINTER TO BOOL;
END_VAR
VAR_OUTPUT
	WERRORID : WORD;
END_VAR
END_METHOD

METHOD HLP_WRITEPARAMETER : BOOL
VAR_INPUT
	PARAMETER : DINT;
	PLRVALUE : POINTER TO LREAL;
END_VAR
VAR_OUTPUT
	WERRORID : WORD;
END_VAR
END_METHOD

METHOD AFTERREADINPUTS : INT
END_METHOD

METHOD AFTERWRITEOUTPUTS : INT
END_METHOD

METHOD BEFOREREADINPUTS : INT
END_METHOD

METHOD BEFOREWRITEOUTPUTS : INT
END_METHOD

METHOD CALCAFTERREADINPUTS : INT
END_METHOD

METHOD CALCAFTERWRITEOUTPUTS : INT
END_METHOD

METHOD CALCBEFOREREADINPUTS : INT
END_METHOD

METHOD CALCBEFOREWRITEOUTPUTS : INT
END_METHOD

METHOD FB_EXIT : BOOL
VAR_INPUT
	BINCOPYCODE : BOOL;
END_VAR
END_METHOD

METHOD INITFORSIMULATIONMODE : BOOL
VAR_INPUT
	WMODULETYPE : UINT;
	DWINSTANCE : UDINT;
	PCONNECTOR : POINTER TO IoConfigConnector;
END_VAR
END_METHOD

METHOD INITIALIZE : UDINT
VAR_INPUT
	WMODULETYPE : UINT;
	DWINSTANCE : UDINT;
	PCONNECTOR : POINTER TO IoConfigConnector;
END_VAR
END_METHOD

METHOD IODRVREADPARAMETER : UDINT
VAR_INPUT
	PCONNECTOR : POINTER TO IoConfigConnector;
	PPARAMETER : POINTER TO IoConfigParameter;
	PDATA : POINTER TO BYTE;
	DWBITSIZE : DWORD;
	DWBITOFFSET : DWORD;
END_VAR
END_METHOD

METHOD IODRVUPDATECONFIGURATION : UDINT
VAR_INPUT
	PCONNECTORLIST : POINTER TO IoConfigConnector;
	NCOUNT : DINT;
END_VAR
END_METHOD

METHOD IODRVUPDATEMAPPING : UDINT
VAR_INPUT
	PTASKMAPLIST : POINTER TO IoConfigTaskMap;
	NCOUNT : DINT;
END_VAR
END_METHOD

METHOD IODRVWRITEPARAMETER : UDINT
VAR_INPUT
	PCONNECTOR : POINTER TO IoConfigConnector;
	PPARAMETER : POINTER TO IoConfigParameter;
	PDATA : POINTER TO BYTE;
	DWBITSIZE : DWORD;
	DWBITOFFSET : DWORD;
END_VAR
END_METHOD

METHOD FB_INIT : BOOL
VAR_INPUT
	BINITRETAINS : BOOL;
	BINCOPYCODE : BOOL;
END_VAR
END_METHOD

METHOD FUNCTIONSUPPORTEDBYAXIS : BOOL
VAR_INPUT
	FUNID : L_MC1P_AxisFunction;
	XORIGINDEVICE : BOOL;
END_VAR
END_METHOD

METHOD GETDELAYFORFASTOUTPUTCALCULATION : LREAL
VAR_INPUT
	EVALUESOURCE : MC_SOURCE;
END_VAR
END_METHOD

METHOD GETINDEXOFENCODERCRC : WORD
END_METHOD

METHOD GETINDEXOFERRORCODE : DINT
END_METHOD

METHOD GETINDEXOFPOSCTRLADAPTVALUE
VAR_INPUT
	WSELECTION : WORD;
END_VAR
VAR_OUTPUT
	WINDEX : WORD;
	BYSUBINDEX : BYTE;
	BYSIZE : BYTE;
END_VAR
END_METHOD

METHOD GETINDEXOFSPEEDCTRLADAPTVALUE
VAR_INPUT
	WSELECTION : WORD;
END_VAR
VAR_OUTPUT
	WINDEX : WORD;
	BYSUBINDEX : BYTE;
	BYSIZE : BYTE;
END_VAR
END_METHOD

METHOD GETMAGNETISATIONFINISHED : BOOL
END_METHOD

METHOD GETMAXTORQUE : LREAL
END_METHOD

METHOD GETREFERENCETORQUE : LREAL
END_METHOD

METHOD GETTPDELAYFORFASTINPUTCALCULATION : LREAL
END_METHOD

METHOD GETVPPMAXVALUE : LREAL
END_METHOD

METHOD SETSPEEDCTRLLIMITATION : BOOL
VAR_INPUT
	XLIMIT : BOOL;
END_VAR
END_METHOD

METHOD SUPPORTLIMITSPEEDCONTROLLER : BOOL
VAR_OUTPUT
	WINDEX : WORD;
	BYSUBINDEX : BYTE;
	BYSIZE : BYTE;
END_VAR
END_METHOD

METHOD SUPPORTMFE : BOOL
END_METHOD

METHOD CALCDISTANCE : LREAL
VAR_INPUT
	LRROUNDSACT : LREAL;
	LRROUNDSSET : LREAL;
	LRPOSACT : LREAL;
	LRPOSSET : LREAL;
END_VAR
VAR_IN_OUT
	AXIS : AXIS_REF;
END_VAR
END_METHOD

METHOD CALCTARGETPOS : LREAL
VAR_INPUT
	LRROUNDSACT : LREAL;
	LRROUNDSSET : LREAL;
	LRPOSACT : LREAL;
	LRPOSSET : LREAL;
END_VAR
VAR_OUTPUT
	EDIR : MC_DIRECTION;
END_VAR
VAR_IN_OUT
	AXIS : AXIS_REF;
END_VAR
END_METHOD

METHOD SETPOSRECOVERYDATA
VAR_INPUT
	XACTIVATE : BOOL;
	LRVEL : LREAL;
	LRACC : LREAL;
	LRDEC : LREAL;
	LRJERK : LREAL;
END_VAR
END_METHOD

(* ---- AXIS_REF_9400HL.pou ---- *)
FUNCTION_BLOCK AXIS_REF_9400HL EXTENDS _AXIS_REF_9400HL
VAR
	PARA_AXIS_REF_9400HL : L_MC1P_ParaInterface_AXIS_REF_9400HL;
END_VAR
END_FUNCTION_BLOCK

METHOD FB_INIT : BOOL
VAR_INPUT
	BINITRETAINS : BOOL;
	BINCOPYCODE : BOOL;
END_VAR
END_METHOD

(* ---- AXIS_REF_9400HL_CAN.pou ---- *)
FUNCTION_BLOCK AXIS_REF_9400HL_CAN EXTENDS _AXIS_REF_9400HL_CAN
VAR
	PARA_AXIS_REF_9400HL_CAN : L_MC1P_ParaInterface_AXIS_REF_9400HL_CAN;
END_VAR
END_FUNCTION_BLOCK

METHOD FB_INIT : BOOL
VAR_INPUT
	BINITRETAINS : BOOL;
	BINCOPYCODE : BOOL;
END_VAR
END_METHOD

(* ---- AXIS_REF_ENC_BPB.pou ---- *)
FUNCTION_BLOCK AXIS_REF_ENC_BPB EXTENDS _AXIS_REF_ENC_BPB
VAR
	PARA_AXIS_REF_ENC_BPB : L_MC1P_ParaInterface_AXIS_REF_ENC_BPB;
END_VAR
END_FUNCTION_BLOCK

METHOD FB_INIT : BOOL
VAR_INPUT
	BINITRETAINS : BOOL;
	BINCOPYCODE : BOOL;
END_VAR
END_METHOD

(* ---- AXIS_REF_ENC_FREE.pou ---- *)
FUNCTION_BLOCK AXIS_REF_ENC_FREE EXTENDS _AXIS_REF_ENC_FREE
VAR
	PARA_AXIS_REF_ENC_FREE : L_MC1P_ParaInterface_AXIS_REF_ENC_FREE;
END_VAR
END_FUNCTION_BLOCK

METHOD FB_INIT : BOOL
VAR_INPUT
	BINITRETAINS : BOOL;
	BINCOPYCODE : BOOL;
END_VAR
END_METHOD

(* ---- AXIS_REF_ENC_I500_ECAT.pou ---- *)
FUNCTION_BLOCK AXIS_REF_ENC_I500_ECAT EXTENDS _AXIS_REF_ENC_i500_ECAT
VAR
	PARA_AXIS_REF_ENC_I500_ECAT : L_MC1P_ParaInterface_AXIS_REF_ENC_i500_ECAT;
END_VAR
END_FUNCTION_BLOCK

METHOD FB_INIT : BOOL
VAR_INPUT
	BINITRETAINS : BOOL;
	BINCOPYCODE : BOOL;
END_VAR
END_METHOD

(* ---- AXIS_REF_ENC_I900_DRIVE.pou ---- *)
FUNCTION_BLOCK AXIS_REF_ENC_I900_DRIVE EXTENDS _AXIS_REF_ENC_i900_Target
VAR
	PARA_AXIS_REF_ENC_I900_DRIVE : L_MC1P_ParaInterface_AXIS_REF_ENC_i900_DRIVE;
END_VAR
END_FUNCTION_BLOCK

METHOD FB_INIT : BOOL
VAR_INPUT
	BINITRETAINS : BOOL;
	BINCOPYCODE : BOOL;
END_VAR
END_METHOD

(* ---- AXIS_REF_ENC_I900_DRIVE_CIA.pou ---- *)
FUNCTION_BLOCK AXIS_REF_ENC_I900_DRIVE_CIA EXTENDS _AXIS_REF_ENC_i900_CiA
VAR
	PARA_AXIS_REF_ENC_I900_DRIVE_CIA : L_MC1P_ParaInterface_AXIS_REF_ENC_i900_DRIVE_CIA;
END_VAR
END_FUNCTION_BLOCK

METHOD FB_INIT : BOOL
VAR_INPUT
	BINITRETAINS : BOOL;
	BINCOPYCODE : BOOL;
END_VAR
END_METHOD

(* ---- AXIS_REF_ENC_I900_ECAT.pou ---- *)
FUNCTION_BLOCK AXIS_REF_ENC_I900_ECAT EXTENDS _AXIS_REF_ENC_i900_ECAT
VAR
	PARA_AXIS_REF_ENC_I900_ECAT : L_MC1P_ParaInterface_AXIS_REF_ENC_i900_ECAT;
END_VAR
END_FUNCTION_BLOCK

METHOD FB_INIT : BOOL
VAR_INPUT
	BINITRETAINS : BOOL;
	BINCOPYCODE : BOOL;
END_VAR
END_METHOD

(* ---- AXIS_REF_ENC_IO_ETC.pou ---- *)
FUNCTION_BLOCK AXIS_REF_ENC_IO_ETC EXTENDS _AXIS_REF_ENC_IO_ETC
VAR
	PARA_AXIS_REF_ENC_IO_ETC : L_MC1P_ParaInterface_AXIS_REF_ENC_IO_ETC;
END_VAR
END_FUNCTION_BLOCK

METHOD FB_INIT : BOOL
VAR_INPUT
	BINITRETAINS : BOOL;
	BINCOPYCODE : BOOL;
END_VAR
END_METHOD

(* ---- AXIS_REF_ENC_UNIVERSAL.pou ---- *)
FUNCTION_BLOCK AXIS_REF_ENC_UNIVERSAL EXTENDS _AXIS_REF_Enc_Universal
VAR
	PARA_AXIS_REF_ENC_UNIVERSAL : L_MC1P_ParaInterface_AXIS_REF_ENC_UNIVERSAL;
END_VAR
END_FUNCTION_BLOCK

METHOD FB_INIT : BOOL
VAR_INPUT
	BINITRETAINS : BOOL;
	BINCOPYCODE : BOOL;
END_VAR
END_METHOD

(* ---- AXIS_REF_GENERIC.pou ---- *)
FUNCTION_BLOCK AXIS_REF_GENERIC EXTENDS _AXIS_REF_GENERIC
VAR
	PARA_AXIS_REF_GENERIC : L_MC1P_ParaInterface_AXIS_REF_GENERIC;
END_VAR
END_FUNCTION_BLOCK

METHOD FB_INIT : BOOL
VAR_INPUT
	BINITRETAINS : BOOL;
	BINCOPYCODE : BOOL;
END_VAR
END_METHOD

(* ---- AXIS_REF_I500_CAN.pou ---- *)
FUNCTION_BLOCK AXIS_REF_I500_CAN EXTENDS _AXIS_REF_i500_CAN
VAR
	PARA_AXIS_REF_I500_CAN : L_MC1P_ParaInterface_AXIS_REF_i500_CAN;
END_VAR
END_FUNCTION_BLOCK

METHOD FB_INIT : BOOL
VAR_INPUT
	BINITRETAINS : BOOL;
	BINCOPYCODE : BOOL;
END_VAR
END_METHOD

(* ---- AXIS_REF_I500_ETC.pou ---- *)
FUNCTION_BLOCK AXIS_REF_I500_ETC EXTENDS _AXIS_REF_i500_ETC
VAR
	PARA_AXIS_REF_I500_ETC : L_MC1P_ParaInterface_AXIS_REF_i500_ETC;
END_VAR
END_FUNCTION_BLOCK

METHOD FB_INIT : BOOL
VAR_INPUT
	BINITRETAINS : BOOL;
	BINCOPYCODE : BOOL;
END_VAR
END_METHOD

(* ---- AXIS_REF_I700.pou ---- *)
FUNCTION_BLOCK AXIS_REF_I700 EXTENDS _AXIS_REF_i700
VAR
	PARA_AXIS_REF_I700 : L_MC1P_ParaInterface_AXIS_REF_i700;
END_VAR
END_FUNCTION_BLOCK

METHOD FB_INIT : BOOL
VAR_INPUT
	BINITRETAINS : BOOL;
	BINCOPYCODE : BOOL;
END_VAR
END_METHOD

(* ---- AXIS_REF_I700_SLOT1.pou ---- *)
FUNCTION_BLOCK AXIS_REF_I700_SLOT1 EXTENDS _AXIS_REF_i700_SLOT1
VAR
	PARA_AXIS_REF_I700_SLOT1 : L_MC1P_ParaInterface_AXIS_REF_i700_SLOT1;
END_VAR
END_FUNCTION_BLOCK

METHOD FB_INIT : BOOL
VAR_INPUT
	BINITRETAINS : BOOL;
	BINCOPYCODE : BOOL;
END_VAR
END_METHOD

(* ---- AXIS_REF_I750.pou ---- *)
FUNCTION_BLOCK AXIS_REF_I750 EXTENDS _AXIS_REF_i750
VAR
	PARA_AXIS_REF_I750 : L_MC1P_ParaInterface_AXIS_REF_i750;
END_VAR
END_FUNCTION_BLOCK

METHOD FB_INIT : BOOL
VAR_INPUT
	BINITRETAINS : BOOL;
	BINCOPYCODE : BOOL;
END_VAR
END_METHOD

(* ---- AXIS_REF_I900.pou ---- *)
FUNCTION_BLOCK AXIS_REF_I900 EXTENDS _AXIS_REF_i900
VAR
	PARA_AXIS_REF_I900 : L_MC1P_ParaInterface_AXIS_REF_i900;
END_VAR
END_FUNCTION_BLOCK

METHOD FB_INIT : BOOL
VAR_INPUT
	BINITRETAINS : BOOL;
	BINCOPYCODE : BOOL;
END_VAR
END_METHOD

(* ---- AXIS_REF_I900_CIAADV.pou ---- *)
FUNCTION_BLOCK AXIS_REF_I900_CIAADV EXTENDS _AXIS_REF_i900_CiaAdv
VAR
	PARA_AXIS_REF_I900_CIAADV : L_MC1P_ParaInterface_AXIS_REF_i900_CiaAdv;
END_VAR
END_FUNCTION_BLOCK

METHOD FB_INIT : BOOL
VAR_INPUT
	BINITRETAINS : BOOL;
	BINCOPYCODE : BOOL;
END_VAR
END_METHOD

(* ---- AXIS_REF_I900_DRIVE.pou ---- *)
FUNCTION_BLOCK AXIS_REF_I900_DRIVE EXTENDS _AXIS_REF_i900_Drive_Target
VAR
	PARA_AXIS_REF_I900_DRIVE : L_MC1P_ParaInterface_AXIS_REF_i900_DRIVE;
END_VAR
END_FUNCTION_BLOCK

METHOD FB_INIT : BOOL
VAR_INPUT
	BINITRETAINS : BOOL;
	BINCOPYCODE : BOOL;
END_VAR
END_METHOD

(* ---- AXIS_REF_I900_DRIVE_CIA.pou ---- *)
FUNCTION_BLOCK AXIS_REF_I900_DRIVE_CIA EXTENDS _AXIS_REF_i900_Drive_CiA
VAR
	PARA_AXIS_REF_I900_DRIVE_CIA : L_MC1P_ParaInterface_AXIS_REF_i900_DRIVE_CIA;
END_VAR
END_FUNCTION_BLOCK

METHOD FB_INIT : BOOL
VAR_INPUT
	BINITRETAINS : BOOL;
	BINCOPYCODE : BOOL;
END_VAR
END_METHOD

(* ---- AXIS_REF_UNIVERSAL.pou ---- *)
FUNCTION_BLOCK AXIS_REF_UNIVERSAL EXTENDS _AXIS_REF_Universal
VAR
	PARA_AXIS_REF_UNIVERSAL : L_MC1P_ParaInterface_AXIS_REF_UNIVERSAL;
END_VAR
END_FUNCTION_BLOCK

METHOD FB_INIT : BOOL
VAR_INPUT
	BINITRETAINS : BOOL;
	BINCOPYCODE : BOOL;
END_VAR
END_METHOD

(* ---- AXIS_REF_VIRTUAL.pou ---- *)
FUNCTION_BLOCK AXIS_REF_VIRTUAL EXTENDS AXIS_REF
VAR
	PARA_AXIS_REF_VIRTUAL : L_MC1P_ParaInterface_AXIS_REF_VIRTUAL;
END_VAR
END_FUNCTION_BLOCK

METHOD FB_INIT : BOOL
VAR_INPUT
	BINITRETAINS : BOOL;
	BINCOPYCODE : BOOL;
END_VAR
END_METHOD

(* ---- AXIS_REF_VIRTUALM_I900.pou ---- *)
FUNCTION_BLOCK AXIS_REF_VIRTUALM_I900 EXTENDS AXIS_REF
VAR
	PARA_AXIS_REF_VIRTUALM_I900 : L_MC1P_ParaInterface_AXIS_REF_VIRTUALM_i900;
END_VAR
END_FUNCTION_BLOCK

METHOD FB_INIT : BOOL
VAR_INPUT
	BINITRETAINS : BOOL;
	BINCOPYCODE : BOOL;
END_VAR
END_METHOD

(* ---- AXIS_REF_VMA.pou ---- *)
FUNCTION_BLOCK AXIS_REF_VMA EXTENDS _AXIS_REF_VMA
VAR
	PARA_AXIS_REF_VMA : L_MC1P_ParaInterface_AXIS_REF_VMA;
END_VAR
END_FUNCTION_BLOCK

METHOD FB_INIT : BOOL
VAR_INPUT
	BINITRETAINS : BOOL;
	BINCOPYCODE : BOOL;
END_VAR
END_METHOD

(* ---- GLOBALTEXTLIST.pou ---- *)
FUNCTION_BLOCK GLOBALTEXTLIST
VAR
	M_TEXTLISTFILE : STRING(255);
	_STNAMESPACE : STRING;
END_VAR
END_FUNCTION_BLOCK

(* ---- IMAGEPOOL.pou ---- *)
FUNCTION_BLOCK IMAGEPOOL
VAR
	M_STNAMESPACE : STRING(80);
	M_STHELPVARID : STRING;
	M_STHELPVARPATH : STRING(255);
	M_STHELP : STRING;
	M_REGISTERIMAGES : BOOL := TRUE;
END_VAR
END_FUNCTION_BLOCK

METHOD FB_INIT : BOOL
VAR_INPUT
	BINITRETAINS : BOOL;
	BINCOPYCODE : BOOL;
END_VAR
END_METHOD

METHOD FB_REINIT : BOOL
END_METHOD

METHOD FB_EXIT : BOOL
VAR_INPUT
	BINCOPYCODE : BOOL;
END_VAR
END_METHOD
